KUKA KRL program: MyProgram_108().src

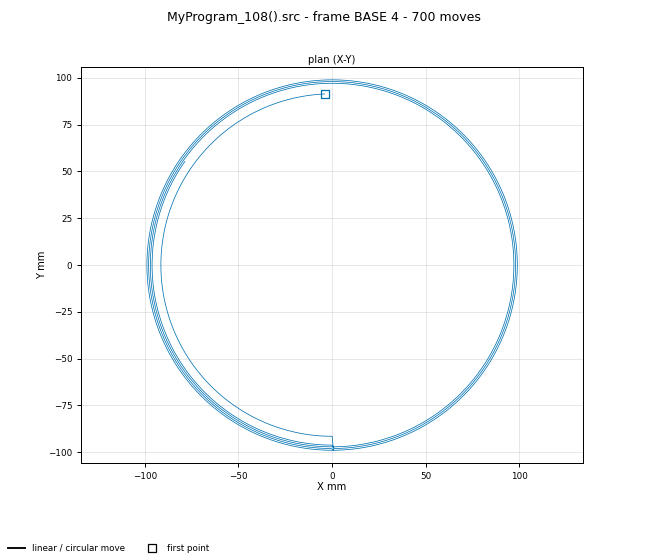
[picture p0: tool path of MyProgram_108().src in frame BASE 4, 700 of 700 moves have a stored position in this frame; points joined in program order, loops and branches not executed]
&ACCESS RVP
&REL 1
&PARAM TEMPLATE = C:\KRC\Roboter\Template\vorgabe
&PARAM EDITMASK = *
DEF MyProgram_108()
; ---- Setting reference (Base) ----
$BASE = BASE_DATA[4]

; --------------------------
; ---- Setting tool (TCP) ----
$TOOL = TOOL_DATA[3]
; --------------------------

$VEL.CP = VEL_APROX_PRINT
Startdeposition()
$VEL.CP = VEL_PRINT
LIN {X -4.0238,Y 91.3698,Z 95,A 87.6224,B 24.9054,C -2.2454,E1 24.992,E2 357.3815} C_DIS
LIN {X -6.9147,Y 91.1973,Z 95,A 89.45,B 24.9054,C -2.2451,E1 24.9869,E2 355.554} C_DIS
LIN {X -9.3244,Y 90.982,Z 95,A 91.0021,B 24.9054,C -2.2455,E1 24.9826,E2 354} C_DIS
LIN {X -12.2843,Y 90.6312,Z 95,A 92.9246,B 24.9054,C -2.2462,E1 24.9773,E2 352.0746} C_DIS
LIN {X -15.2613,Y 90.1762,Z 95,A 94.7056,B 24.9058,C -2.2414,E1 24.9724,E2 350.3032} C_DIS
LIN {X -18.2109,Y 89.6272,Z 95,A 96.5328,B 24.906,C -2.2382,E1 24.9674,E2 348.4816} C_DIS
LIN {X -20.6734,Y 89.0912,Z 95,A 98.1962,B 24.906,C -2.2396,E1 24.9628,E2 346.8129} C_DIS
LIN {X -23.8987,Y 88.2807,Z 95,A 100.2948,B 24.906,C -2.238,E1 24.9572,E2 344.715} C_DIS
LIN {X -26.5206,Y 87.5304,Z 95,A 102.081,B 24.906,C -2.2386,E1 24.9524,E2 342.9244} C_DIS
LIN {X -29.3987,Y 86.6047,Z 95,A 103.8698,B 24.9065,C -2.233,E1 24.9476,E2 341.1456} C_DIS
LIN {X -32.2068,Y 85.6002,Z 95,A 105.7005,B 24.9068,C -2.2294,E1 24.9429,E2 339.3198} C_DIS
LIN {X -34.3185,Y 84.7756,Z 95,A 107.1121,B 24.907,C -2.2272,E1 24.9392,E2 337.9104} C_DIS
LIN {X -36.7249,Y 83.7613,Z 95,A 108.969,B 24.9066,C -2.2318,E1 24.9344,E2 336.038} C_DIS
LIN {X -39.7684,Y 82.3598,Z 95,A 110.9169,B 24.9072,C -2.2238,E1 24.9295,E2 334.1043} C_DIS
LIN {X -42.0959,Y 81.1963,Z 95,A 112.6486,B 24.9072,C -2.2243,E1 24.9252,E2 332.3667} C_DIS
LIN {X -44.3837,Y 79.9673,Z 95,A 114.2579,B 24.9075,C -2.221,E1 24.9213,E2 330.7607} C_DIS
LIN {X -47.031,Y 78.4412,Z 95,A 116.0516,B 24.9081,C -2.2137,E1 24.917,E2 328.9788} C_DIS
LIN {X -48.938,Y 77.2658,Z 95,A 117.4609,B 24.9083,C -2.2113,E1 24.9136,E2 327.5709} C_DIS
LIN {X -50.8158,Y 76.044,Z 95,A 118.8703,B 24.9085,C -2.2088,E1 24.9104,E2 326.1629} C_DIS
LIN {X -52.965,Y 74.5612,Z 95,A 120.6248,B 24.9085,C -2.2093,E1 24.9063,E2 324.4013} C_DIS
LIN {X -55.6722,Y 72.5622,Z 95,A 122.7413,B 24.9088,C -2.2051,E1 24.9016,E2 322.287} C_DIS
LIN {X -58.1699,Y 70.5764,Z 95,A 124.7763,B 24.9091,C -2.2019,E1 24.8972,E2 320.2521} C_DIS
LIN {X -60.5846,Y 68.516,Z 95,A 126.8574,B 24.9091,C -2.2003,E1 24.8928,E2 318.1667} C_DIS
LIN {X -63.0597,Y 66.2451,Z 95,A 128.9712,B 24.9096,C -2.1956,E1 24.8885,E2 316.0552} C_DIS
LIN {X -65.4493,Y 63.8852,Z 95,A 131.0907,B 24.91,C -2.191,E1 24.8843,E2 313.9377} C_DIS
LIN {X -67.7678,Y 61.4204,Z 95,A 133.2194,B 24.9104,C -2.186,E1 24.8803,E2 311.8115} C_DIS
LIN {X -69.9777,Y 58.8902,Z 95,A 135.335,B 24.9108,C -2.181,E1 24.8765,E2 309.6983} C_DIS
LIN {X -72.0929,Y 56.2809,Z 95,A 137.4,B 24.9113,C -2.1742,E1 24.8729,E2 307.6397} C_DIS
LIN {X -73.682,Y 54.1815,Z 95,A 139.0043,B 24.9118,C -2.1684,E1 24.8702,E2 306.0416} C_DIS
LIN {X -75.623,Y 51.4376,Z 95,A 141.012,B 24.9125,C -2.1597,E1 24.8671,E2 304.0448} C_DIS
LIN {X -76.8604,Y 49.5696,Z 95,A 142.4242,B 24.9128,C -2.156,E1 24.8649,E2 302.6342} C_DIS
LIN {X -78.3252,Y 47.2218,Z 95,A 144.3699,B 24.9127,C -2.1575,E1 24.862,E2 300.6749} C_DIS
LIN {X -79.9567,Y 44.4027,Z 95,A 146.4407,B 24.9131,C -2.1526,E1 24.8592,E2 298.6051} C_DIS
LIN {X -81.3588,Y 41.778,Z 95,A 148.0983,B 24.914,C -2.1408,E1 24.8571,E2 296.9667} C_DIS
LIN {X -82.3563,Y 39.7757,Z 95,A 149.6193,B 24.914,C -2.1403,E1 24.8552,E2 295.4387} C_DIS
LIN {X -83.7601,Y 36.7275,Z 95,A 151.7374,B 24.9146,C -2.1345,E1 24.8528,E2 293.323} C_DIS
LIN {X -84.9155,Y 33.9747,Z 95,A 153.5097,B 24.9152,C -2.1258,E1 24.8509,E2 291.5616} C_DIS
LIN {X -85.8476,Y 31.5416,Z 95,A 155.2735,B 24.9153,C -2.1248,E1 24.8492,E2 289.7902} C_DIS
LIN {X -86.8443,Y 28.6883,Z 95,A 157.2742,B 24.9155,C -2.1221,E1 24.8474,E2 287.7845} C_DIS
LIN {X -87.8446,Y 25.4609,Z 95,A 159.1895,B 24.9165,C -2.1094,E1 24.8459,E2 285.8885} C_DIS
LIN {X -88.5337,Y 22.9445,Z 95,A 160.8359,B 24.9169,C -2.1047,E1 24.8447,E2 284.2438} C_DIS
LIN {X -89.154,Y 20.4015,Z 95,A 162.5816,B 24.9171,C -2.1027,E1 24.8435,E2 282.4927} C_DIS
LIN {X -89.7713,Y 17.4864,Z 95,A 164.4831,B 24.9175,C -2.0978,E1 24.8425,E2 280.5916} C_DIS
LIN {X -90.2986,Y 14.5298,Z 95,A 166.4559,B 24.9177,C -2.0945,E1 24.8416,E2 278.6149} C_DIS
LIN {X -90.677,Y 11.931,Z 95,A 167.9188,B 24.9186,C -2.0838,E1 24.841,E2 277.1689} C_DIS
LIN {X -90.9812,Y 9.3323,Z 95,A 169.7863,B 24.9184,C -2.0854,E1 24.8405,E2 275.2863} C_DIS
LIN {X -91.2368,Y 6.3646,Z 95,A 171.5613,B 24.9191,C -2.0766,E1 24.8401,E2 273.5216} C_DIS
LIN {X -91.3974,Y 3.3826,Z 95,A 173.3436,B 24.9198,C -2.068,E1 24.8399,E2 271.7493} C_DIS
LIN {X -91.4559,Y 0.6849,Z 95,A 175.1899,B 24.9198,C -2.0673,E1 24.8398,E2 269.8934} C_DIS
LIN {X -91.4213,Y -2.6095,Z 95,A 177.226,B 24.9204,C -2.0598,E1 24.8398,E2 267.8629} C_DIS
LIN {X -91.2891,Y -5.5881,Z 95,A 178.9966,B 24.9211,C -2.0509,E1 24.8402,E2 266.1029} C_DIS
LIN {X -91.092,Y -8.1813,Z 95,A -179.2539,B 24.9212,C -2.0494,E1 24.8406,E2 264.3466} C_DIS
LIN {X -90.7722,Y -11.1963,Z 95,A -177.45,B 24.9219,C -2.0405,E1 24.8411,E2 262.5531} C_DIS
LIN {X -90.4152,Y -13.7756,Z 95,A -175.6959,B 24.922,C -2.0391,E1 24.8418,E2 260.7919} C_DIS
LIN {X -89.8677,Y -16.9857,Z 95,A -173.7041,B 24.9226,C -2.0313,E1 24.8428,E2 258.8069} C_DIS
LIN {X -89.3965,Y -19.3113,Z 95,A -172.2569,B 24.9231,C -2.0255,E1 24.8436,E2 257.365} C_DIS
LIN {X -88.8068,Y -21.8634,Z 95,A -170.388,B 24.9229,C -2.0274,E1 24.8449,E2 255.4806} C_DIS
LIN {X -87.9436,Y -25.1114,Z 95,A -168.2536,B 24.9233,C -2.0219,E1 24.8465,E2 253.3469} C_DIS
LIN {X -86.9741,Y -28.287,Z 95,A -166.3203,B 24.9242,C -2.0112,E1 24.8481,E2 251.428} C_DIS
LIN {X -85.9537,Y -31.2506,Z 95,A -164.3287,B 24.9245,C -2.0062,E1 24.8499,E2 249.4369} C_DIS
LIN {X -84.7924,Y -34.2772,Z 95,A -162.3782,B 24.9252,C -1.9979,E1 24.8519,E2 247.4954} C_DIS
LIN {X -83.7612,Y -36.725,Z 95,A -160.48,B 24.925,C -2.0003,E1 24.854,E2 245.581} C_DIS
LIN {X -82.3569,Y -39.7745,Z 95,A -158.5243,B 24.9258,C -1.9899,E1 24.8563,E2 243.6396} C_DIS
LIN {X -81.1905,Y -42.1074,Z 95,A -156.7702,B 24.9258,C -1.989,E1 24.8586,E2 241.8781} C_DIS
LIN {X -79.9424,Y -44.4283,Z 95,A -155.1647,B 24.9263,C -1.9832,E1 24.8607,E2 240.278} C_DIS
LIN {X -78.4484,Y -47.019,Z 95,A -153.3895,B 24.9269,C -1.9752,E1 24.8632,E2 238.5128} C_DIS
LIN {X -77.2616,Y -48.9446,Z 95,A -151.9685,B 24.9271,C -1.9716,E1 24.8653,E2 237.093} C_DIS
LIN {X -76.0454,Y -50.8137,Z 95,A -150.5605,B 24.9274,C -1.9684,E1 24.8675,E2 235.6856} C_DIS
LIN {X -74.5698,Y -52.9529,Z 95,A -148.8116,B 24.9274,C -1.9681,E1 24.8703,E2 233.9288} C_DIS
LIN {X -72.467,Y -55.7958,Z 95,A -146.5187,B 24.9276,C -1.9651,E1 24.8742,E2 231.6319} C_DIS
LIN {X -70.3336,Y -58.4621,Z 95,A -144.434,B 24.9281,C -1.9584,E1 24.8778,E2 229.5536} C_DIS
LIN {X -68.1382,Y -61.0067,Z 95,A -142.3198,B 24.9284,C -1.9539,E1 24.8817,E2 227.4405} C_DIS
LIN {X -65.8506,Y -63.4691,Z 95,A -140.204,B 24.9287,C -1.9496,E1 24.8858,E2 225.3258} C_DIS
LIN {X -63.474,Y -65.8459,Z 95,A -138.0877,B 24.929,C -1.9456,E1 24.89,E2 223.2102} C_DIS
LIN {X -60.9908,Y -68.1525,Z 95,A -135.9582,B 24.9293,C -1.9415,E1 24.8944,E2 221.0817} C_DIS
LIN {X -58.4524,Y -70.3416,Z 95,A -133.8322,B 24.9296,C -1.9384,E1 24.8989,E2 218.9551} C_DIS
LIN {X -55.8153,Y -72.4519,Z 95,A -131.7259,B 24.9299,C -1.9342,E1 24.9035,E2 216.8509} C_DIS
LIN {X -53.5848,Y -74.1188,Z 95,A -129.9248,B 24.9299,C -1.933,E1 24.9076,E2 215.0463} C_DIS
LIN {X -51.4624,Y -75.6062,Z 95,A -128.4555,B 24.9305,C -1.9255,E1 24.9109,E2 213.59} C_DIS
LIN {X -49.6142,Y -76.8318,Z 95,A -127.0642,B 24.9306,C -1.9234,E1 24.9142,E2 212.1992} C_DIS
LIN {X -47.6627,Y -78.0572,Z 95,A -125.4981,B 24.9306,C -1.9252,E1 24.9179,E2 210.624} C_DIS
LIN {X -45.086,Y -79.5751,Z 95,A -123.5397,B 24.9306,C -1.9252,E1 24.9227,E2 208.6596} C_DIS
LIN {X -42.7806,Y -80.8361,Z 95,A -122.0791,B 24.9311,C -1.9171,E1 24.9262,E2 207.2143} C_DIS
LIN {X -40.6274,Y -81.9393,Z 95,A -120.4471,B 24.931,C -1.919,E1 24.9303,E2 205.5733} C_DIS
LIN {X -38.0993,Y -83.1467,Z 95,A -118.6241,B 24.931,C -1.9192,E1 24.935,E2 203.7454} C_DIS
LIN {X -35.3431,Y -84.3536,Z 95,A -116.8551,B 24.9314,C -1.9134,E1 24.9395,E2 201.9859} C_DIS
LIN {X -32.8352,Y -85.3622,Z 95,A -115.0915,B 24.9314,C -1.9141,E1 24.9441,E2 200.2169} C_DIS
LIN {X -30.4684,Y -86.2342,Z 95,A -113.6232,B 24.9317,C -1.909,E1 24.9479,E2 198.7577} C_DIS
LIN {X -27.9724,Y -87.0759,Z 95,A -111.9226,B 24.9317,C -1.9094,E1 24.9524,E2 197.0531} C_DIS
LIN {X -25.1205,Y -87.9411,Z 95,A -109.9953,B 24.9317,C -1.9101,E1 24.9576,E2 195.1209} C_DIS
LIN {X -21.8609,Y -88.8075,Z 95,A -107.8812,B 24.9317,C -1.9089,E1 24.9633,E2 193.0065} C_DIS
LIN {X -18.9546,Y -89.4743,Z 95,A -105.9637,B 24.9317,C -1.9097,E1 24.9686,E2 191.0848} C_DIS
LIN {X -15.8541,Y -90.0744,Z 95,A -104.121,B 24.932,C -1.9045,E1 24.9736,E2 189.2526} C_DIS
LIN {X -13.1259,Y -90.5119,Z 95,A -102.2258,B 24.9316,C -1.9095,E1 24.9789,E2 187.3437} C_DIS
LIN {X -9.6461,Y -90.9483,Z 95,A -100.1452,B 24.9319,C -1.9053,E1 24.9846,E2 185.2718} C_DIS
LIN {X -6.6432,Y -91.218,Z 95,A -98.113,B 24.9316,C -1.9101,E1 24.9903,E2 183.2274} C_DIS
LIN {X -3.0457,Y -91.4079,Z 95,A -95.8652,B 24.9316,C -1.9101,E1 24.9966,E2 180.9792} C_DIS
LIN {X 0.0472,Y -91.4598,Z 95,A -93.9773,B 24.9317,C -1.9087,E1 25.0018,E2 179.0946} C_DIS
LIN {X 0.0472,Y -91.4598,Z 95,A -93.9773,B 24.9317,C -1.9087,E1 25.0018,E2 179.0946} C_DIS
Enddeposition()
LIN {X 0.6782,Y -98.9101,Z 96,A -93.6566,B 24.9403,C -1.7848,E1 25.0019,E2 179.0676} C_DIS
Startdeposition()
$VEL.CP = VEL_PRINT
LIN {X 3.095,Y -98.8665,Z 96,A -92.0066,B 24.9396,C -1.7945,E1 25.0066,E2 177.3949} C_DIS
LIN {X 6.0657,Y -98.7307,Z 96,A -90.1754,B 24.9393,C -1.7993,E1 25.0117,E2 175.5531} C_DIS
LIN {X 9.2855,Y -98.4783,Z 96,A -88.4513,B 24.9396,C -1.7947,E1 25.0165,E2 173.8407} C_DIS
LIN {X 12.1085,Y -98.1729,Z 96,A -86.8644,B 24.9397,C -1.7935,E1 25.0209,E2 172.2578} C_DIS
LIN {X 15.0538,Y -97.7627,Z 96,A -85.1441,B 24.9397,C -1.7947,E1 25.0256,E2 170.5364} C_DIS
LIN {X 17.5683,Y -97.3423,Z 96,A -83.58,B 24.9393,C -1.7991,E1 25.03,E2 168.9634} C_DIS
LIN {X 21.0203,Y -96.6557,Z 96,A -81.6027,B 24.9393,C -1.7986,E1 25.0353,E2 166.9899} C_DIS
LIN {X 24.0348,Y -95.9524,Z 96,A -79.6458,B 24.9388,C -1.8066,E1 25.0407,E2 165.0169} C_DIS
LIN {X 26.9078,Y -95.1848,Z 96,A -78.0952,B 24.9391,C -1.8019,E1 25.0448,E2 163.4799} C_DIS
LIN {X 29.8735,Y -94.298,Z 96,A -76.1387,B 24.9386,C -1.8102,E1 25.0501,E2 161.5073} C_DIS
LIN {X 32.909,Y -93.2802,Z 96,A -74.3585,B 24.9386,C -1.8097,E1 25.0548,E2 159.7317} C_DIS
LIN {X 36.1079,Y -92.089,Z 96,A -72.5177,B 24.9388,C -1.8072,E1 25.0596,E2 157.9009} C_DIS
LIN {X 38.357,Y -91.1751,Z 96,A -71.0343,B 24.9384,C -1.8122,E1 25.0634,E2 156.4091} C_DIS
LIN {X 41.1919,Y -89.932,Z 96,A -69.129,B 24.938,C -1.8193,E1 25.0683,E2 154.4918} C_DIS
LIN {X 43.8758,Y -88.6515,Z 96,A -67.6123,B 24.9383,C -1.8141,E1 25.0721,E2 152.9914} C_DIS
LIN {X 46.0382,Y -87.548,Z 96,A -66.1791,B 24.9381,C -1.8175,E1 25.0756,E2 151.554} C_DIS
LIN {X 48.7559,Y -86.0662,Z 96,A -64.4251,B 24.938,C -1.8191,E1 25.0799,E2 149.8014} C_DIS
LIN {X 51.32,Y -84.5602,Z 96,A -62.677,B 24.9377,C -1.8233,E1 25.0841,E2 148.0487} C_DIS
LIN {X 53.9418,Y -82.9145,Z 96,A -60.9235,B 24.9376,C -1.8252,E1 25.0882,E2 146.2965} C_DIS
LIN {X 56.4088,Y -81.2541,Z 96,A -59.1765,B 24.9373,C -1.8296,E1 25.0923,E2 144.5449} C_DIS
LIN {X 58.9247,Y -79.4507,Z 96,A -57.4236,B 24.9371,C -1.8318,E1 25.0962,E2 142.7932} C_DIS
LIN {X 61.2852,Y -77.6421,Z 96,A -55.7092,B 24.9369,C -1.8352,E1 25.1,E2 141.077} C_DIS
LIN {X 63.2658,Y -76.0369,Z 96,A -54.1499,B 24.9364,C -1.8417,E1 25.1034,E2 139.5082} C_DIS
LIN {X 65.5606,Y -74.0694,Z 96,A -52.5233,B 24.9364,C -1.8408,E1 25.1068,E2 137.8902} C_DIS
LIN {X 67.7207,Y -72.0977,Z 96,A -50.812,B 24.9362,C -1.8455,E1 25.1103,E2 136.1747} C_DIS
LIN {X 69.4696,Y -70.414,Z 96,A -49.3807,B 24.9359,C -1.8499,E1 25.1132,E2 134.7391} C_DIS
LIN {X 71.6402,Y -68.2071,Z 96,A -47.4301,B 24.9351,C -1.8605,E1 25.117,E2 132.7717} C_DIS
LIN {X 73.6644,Y -66.0131,Z 96,A -45.9132,B 24.9354,C -1.8565,E1 25.1198,E2 131.271} C_DIS
LIN {X 75.2548,Y -64.1941,Z 96,A -44.5178,B 24.9352,C -1.86,E1 25.1224,E2 129.8737} C_DIS
LIN {X 76.8842,Y -62.2333,Z 96,A -42.96,B 24.9347,C -1.8671,E1 25.1252,E2 128.3064} C_DIS
LIN {X 78.7216,Y -59.8952,Z 96,A -41.1378,B 24.934,C -1.8757,E1 25.1283,E2 126.4725} C_DIS
LIN {X 80.485,Y -57.5007,Z 96,A -39.5926,B 24.9342,C -1.8733,E1 25.1308,E2 124.9403} C_DIS
LIN {X 82.2463,Y -54.9552,Z 96,A -37.6432,B 24.9334,C -1.8846,E1 25.1339,E2 122.9741} C_DIS
LIN {X 84.1104,Y -52.0554,Z 96,A -35.8438,B 24.9336,C -1.8824,E1 25.1365,E2 121.189} C_DIS
LIN {X 85.7335,Y -49.3349,Z 96,A -34.0023,B 24.9332,C -1.8879,E1 25.1391,E2 119.3437} C_DIS
LIN {X 87.2368,Y -46.6291,Z 96,A -32.2525,B 24.9329,C -1.8914,E1 25.1415,E2 117.5948} C_DIS
LIN {X 88.5134,Y -44.1543,Z 96,A -30.5576,B 24.9324,C -1.8995,E1 25.1436,E2 115.8899} C_DIS
LIN {X 89.932,Y -41.1919,Z 96,A -28.5607,B 24.9317,C -1.909,E1 25.146,E2 113.8814} C_DIS
LIN {X 91.1751,Y -38.357,Z 96,A -26.8891,B 24.9317,C -1.9096,E1 25.1478,E2 112.2174} C_DIS
LIN {X 92.4821,Y -35.089,Z 96,A -24.9212,B 24.9314,C -1.9131,E1 25.1498,E2 110.2523} C_DIS
LIN {X 93.5365,Y -32.1787,Z 96,A -22.9733,B 24.9305,C -1.9249,E1 25.1517,E2 108.2876} C_DIS
LIN {X 94.4597,Y -29.3519,Z 96,A -21.4616,B 24.9308,C -1.9218,E1 25.1529,E2 106.7917} C_DIS
LIN {X 95.255,Y -26.6598,Z 96,A -19.8173,B 24.9303,C -1.9277,E1 25.1542,E2 105.143} C_DIS
LIN {X 95.9524,Y -24.0348,Z 96,A -18.0851,B 24.9295,C -1.939,E1 25.1554,E2 103.3939} C_DIS
LIN {X 96.6557,Y -21.0203,Z 96,A -16.4138,B 24.9295,C -1.9399,E1 25.1564,E2 101.7304} C_DIS
LIN {X 97.3423,Y -17.5683,Z 96,A -14.3925,B 24.929,C -1.9457,E1 25.1575,E2 99.7071} C_DIS
LIN {X 97.8462,Y -14.5141,Z 96,A -12.4852,B 24.9283,C -1.956,E1 25.1583,E2 97.7867} C_DIS
LIN {X 98.3141,Y -10.9028,Z 96,A -10.4044,B 24.9279,C -1.9617,E1 25.159,E2 95.7048} C_DIS
LIN {X 98.6053,Y -7.8211,Z 96,A -8.7334,B 24.9278,C -1.9626,E1 25.1594,E2 94.0416} C_DIS
LIN {X 98.8211,Y -4.3081,Z 96,A -6.7984,B 24.9276,C -1.965,E1 25.1597,E2 92.1125} C_DIS
LIN {X 98.8993,Y -1.7598,Z 96,A -5.2454,B 24.927,C -1.9728,E1 25.1597,E2 90.5502} C_DIS
LIN {X 98.8993,Y 1.7598,Z 96,A -3.2752,B 24.9267,C -1.9766,E1 25.1597,E2 88.5828} C_DIS
LIN {X 98.7977,Y 4.8536,Z 96,A -1.3274,B 24.9259,C -1.9886,E1 25.1595,E2 86.6183} C_DIS
LIN {X 98.5956,Y 7.9425,Z 96,A 0.3785,B 24.9257,C -1.9908,E1 25.1592,E2 84.9173} C_DIS
LIN {X 98.2506,Y 11.4452,Z 96,A 2.3109,B 24.9255,C -1.993,E1 25.1586,E2 82.9911} C_DIS
LIN {X 97.8462,Y 14.5141,Z 96,A 4.2589,B 24.9246,C -2.0049,E1 25.1578,E2 81.0266} C_DIS
LIN {X 97.3423,Y 17.5683,Z 96,A 5.9301,B 24.9246,C -2.0056,E1 25.157,E2 79.3634} C_DIS
LIN {X 96.6557,Y 21.0203,Z 96,A 7.8978,B 24.9243,C -2.0091,E1 25.1559,E2 77.399} C_DIS
LIN {X 95.9524,Y 24.0348,Z 96,A 9.8459,B 24.9234,C -2.0208,E1 25.1546,E2 75.4345} C_DIS
LIN {X 95.1516,Y 27.0249,Z 96,A 11.5174,B 24.9234,C -2.0215,E1 25.1534,E2 73.7712} C_DIS
LIN {X 94.298,Y 29.8735,Z 96,A 13.1393,B 24.9233,C -2.0226,E1 25.152,E2 72.1558} C_DIS
LIN {X 93.3556,Y 32.6939,Z 96,A 14.8826,B 24.9228,C -2.0286,E1 25.1505,E2 70.4081} C_DIS
LIN {X 92.2887,Y 35.5997,Z 96,A 16.6325,B 24.9226,C -2.0321,E1 25.1487,E2 68.6598} C_DIS
LIN {X 91.1751,Y 38.357,Z 96,A 18.3438,B 24.9222,C -2.0367,E1 25.1469,E2 66.9471} C_DIS
LIN {X 90.2064,Y 40.583,Z 96,A 19.7417,B 24.9219,C -2.0404,E1 25.1453,E2 65.5481} C_DIS
LIN {X 89.1832,Y 42.7846,Z 96,A 21.1714,B 24.9216,C -2.0453,E1 25.1436,E2 64.1145} C_DIS
LIN {X 87.8025,Y 45.555,Z 96,A 23.121,B 24.9207,C -2.0564,E1 25.1411,E2 62.149} C_DIS
LIN {X 86.3918,Y 48.1728,Z 96,A 24.7172,B 24.9207,C -2.0561,E1 25.139,E2 60.5618} C_DIS
LIN {X 84.8438,Y 50.8534,Z 96,A 26.616,B 24.92,C -2.0651,E1 25.1363,E2 58.6517} C_DIS
LIN {X 83.2095,Y 53.4823,Z 96,A 28.2889,B 24.92,C -2.0651,E1 25.1338,E2 56.9873} C_DIS
LIN {X 81.2541,Y 56.4088,Z 96,A 30.2269,B 24.92,C -2.0663,E1 25.1308,E2 55.0559} C_DIS
LIN {X 79.8328,Y 58.4028,Z 96,A 31.664,B 24.9196,C -2.0705,E1 25.1284,E2 53.6157} C_DIS
LIN {X 77.9807,Y 60.8567,Z 96,A 33.4093,B 24.9194,C -2.0734,E1 25.1255,E2 51.8718} C_DIS
LIN {X 76.4637,Y 62.7522,Z 96,A 35.0079,B 24.9185,C -2.0843,E1 25.1226,E2 50.255} C_DIS
LIN {X 74.5415,Y 65.0211,Z 96,A 36.5222,B 24.9189,C -2.0801,E1 25.1199,E2 48.7574} C_DIS
LIN {X 72.9233,Y 66.8308,Z 96,A 37.9536,B 24.9185,C -2.0843,E1 25.1172,E2 47.3224} C_DIS
LIN {X 70.7978,Y 69.0811,Z 96,A 39.7062,B 24.9184,C -2.0866,E1 25.1138,E2 45.5721} C_DIS
LIN {X 69.0811,Y 70.7978,Z 96,A 41.1059,B 24.9181,C -2.0893,E1 25.111,E2 44.1717} C_DIS
LIN {X 66.9205,Y 72.841,Z 96,A 42.853,B 24.9178,C -2.0938,E1 25.1075,E2 42.4212} C_DIS
LIN {X 64.6098,Y 74.9007,Z 96,A 44.6459,B 24.9175,C -2.0973,E1 25.1037,E2 40.6271} C_DIS
LIN {X 62.7522,Y 76.4637,Z 96,A 46.2064,B 24.9168,C -2.1059,E1 25.1003,E2 39.0522} C_DIS
LIN {X 60.4242,Y 78.314,Z 96,A 47.7948,B 24.917,C -2.1039,E1 25.0968,E2 37.4743} C_DIS
LIN {X 57.9453,Y 80.1678,Z 96,A 49.5086,B 24.917,C -2.1039,E1 25.093,E2 35.7665} C_DIS
LIN {X 55.9604,Y 81.5657,Z 96,A 50.9099,B 24.9168,C -2.1062,E1 25.0898,E2 34.365} C_DIS
LIN {X 53.4823,Y 83.2095,Z 96,A 52.686,B 24.9164,C -2.111,E1 25.0856,E2 32.5833} C_DIS
LIN {X 50.7519,Y 84.9037,Z 96,A 54.527,B 24.9163,C -2.113,E1 25.0812,E2 30.7433} C_DIS
LIN {X 48.1728,Y 86.3918,Z 96,A 56.2909,B 24.916,C -2.1169,E1 25.0769,E2 28.9753} C_DIS
LIN {X 45.555,Y 87.8025,Z 96,A 58.1186,B 24.9155,C -2.1232,E1 25.0724,E2 27.1379} C_DIS
LIN {X 42.7846,Y 89.1832,Z 96,A 59.7968,B 24.9156,C -2.1211,E1 25.0682,E2 25.4692} C_DIS
LIN {X 40.0852,Y 90.4307,Z 96,A 61.425,B 24.9158,C -2.1194,E1 25.0641,E2 23.8489} C_DIS
LIN {X 37.348,Y 91.5931,Z 96,A 63.2176,B 24.9154,C -2.1239,E1 25.0594,E2 22.0498} C_DIS
LIN {X 34.4645,Y 92.7186,Z 96,A 65.1333,B 24.9149,C -2.1302,E1 25.0544,E2 20.1234} C_DIS
LIN {X 31.5458,Y 93.7498,Z 96,A 66.8126,B 24.9151,C -2.1275,E1 25.05,E2 18.4537} C_DIS
LIN {X 28.1905,Y 94.8128,Z 96,A 68.7905,B 24.9151,C -2.1268,E1 25.0447,E2 16.4811} C_DIS
LIN {X 25.2105,Y 95.6502,Z 96,A 70.749,B 24.9146,C -2.1341,E1 25.0394,E2 14.5085} C_DIS
LIN {X 22.3235,Y 96.363,Z 96,A 72.3014,B 24.915,C -2.1288,E1 25.0352,E2 12.9709} C_DIS
LIN {X 19.2977,Y 97.0161,Z 96,A 74.2607,B 24.9145,C -2.1357,E1 25.0298,E2 10.9976} C_DIS
LIN {X 16.2523,Y 97.5706,Z 96,A 75.9419,B 24.9147,C -2.1323,E1 25.0252,E2 9.3264} C_DIS
LIN {X 12.7708,Y 98.0871,Z 96,A 77.9631,B 24.9147,C -2.1321,E1 25.0197,E2 7.3073} C_DIS
LIN {X 9.6955,Y 98.4405,Z 96,A 79.8829,B 24.9143,C -2.137,E1 25.0143,E2 5.3772} C_DIS
LIN {X 6.7319,Y 98.6856,Z 96,A 81.4367,B 24.9148,C -2.1309,E1 25.01,E2 3.8385} C_DIS
LIN {X 3.6409,Y 98.8498,Z 96,A 83.1975,B 24.9149,C -2.1296,E1 25.0051,E2 2.0813} C_DIS
LIN {X 0.6678,Y 98.9127,Z 96,A 84.9532,B 24.9149,C -2.1306,E1 25.0002,E2 0.3236} C_DIS
LIN {X -2.4275,Y 98.887,Z 96,A 86.7149,B 24.9149,C -2.129,E1 24.9953,E2 -1.4344} C_DIS
LIN {X -5.3989,Y 98.7675,Z 96,A 88.4711,B 24.9149,C -2.1297,E1 24.9904,E2 -3.1926} C_DIS
LIN {X -8.4868,Y 98.5521,Z 96,A 90.4345,B 24.9145,C -2.135,E1 24.9849,E2 -5.1695} C_DIS
LIN {X -11.5661,Y 98.2364,Z 96,A 92.1189,B 24.9149,C -2.1301,E1 24.9802,E2 -6.8434} C_DIS
LIN {X -15.0538,Y 97.7627,Z 96,A 94.0705,B 24.9153,C -2.1257,E1 24.9749,E2 -8.786} C_DIS
LIN {X -17.5683,Y 97.3423,Z 96,A 95.64,B 24.9151,C -2.1279,E1 24.9705,E2 -10.3623} C_DIS
LIN {X -21.0203,Y 96.6557,Z 96,A 97.6246,B 24.9154,C -2.1242,E1 24.9651,E2 -12.3406} C_DIS
LIN {X -24.0348,Y 95.9524,Z 96,A 99.5901,B 24.915,C -2.1286,E1 24.9598,E2 -14.3192} C_DIS
LIN {X -26.9078,Y 95.1848,Z 96,A 101.1936,B 24.9155,C -2.1227,E1 24.9555,E2 -15.911} C_DIS
LIN {X -29.8735,Y 94.298,Z 96,A 102.9129,B 24.9159,C -2.118,E1 24.9509,E2 -17.6222} C_DIS
LIN {X -32.1787,Y 93.5365,Z 96,A 104.5242,B 24.9154,C -2.1235,E1 24.9466,E2 -19.2496} C_DIS
LIN {X -35.089,Y 92.4821,Z 96,A 106.2116,B 24.9159,C -2.1175,E1 24.9422,E2 -20.9262} C_DIS
LIN {X -37.8538,Y 91.3872,Z 96,A 107.8487,B 24.9163,C -2.1121,E1 24.938,E2 -22.5541} C_DIS
LIN {X -40.0852,Y 90.4307,Z 96,A 109.32,B 24.9163,C -2.1123,E1 24.9342,E2 -24.0294} C_DIS
LIN {X -42.7846,Y 89.1832,Z 96,A 110.9877,B 24.9167,C -2.1078,E1 24.93,E2 -25.6905} C_DIS
LIN {X -44.9604,Y 88.1064,Z 96,A 112.3992,B 24.9168,C -2.1057,E1 24.9265,E2 -27.1008} C_DIS
LIN {X -47.2161,Y 86.9184,Z 96,A 113.9721,B 24.9168,C -2.1065,E1 24.9226,E2 -28.6801} C_DIS
LIN {X -49.8084,Y 85.4614,Z 96,A 115.8121,B 24.9168,C -2.1075,E1 24.9182,E2 -30.5279} C_DIS
LIN {X -52.4571,Y 83.8595,Z 96,A 117.5015,B 24.9172,C -2.1006,E1 24.9142,E2 -32.2062} C_DIS
LIN {X -54.9552,Y 82.2463,Z 96,A 119.3422,B 24.9172,C -2.1013,E1 24.9099,E2 -34.0547} C_DIS
LIN {X -57.5007,Y 80.485,Z 96,A 121.0324,B 24.9178,C -2.0942,E1 24.906,E2 -35.7337} C_DIS
LIN {X -59.8952,Y 78.7216,Z 96,A 122.8738,B 24.9178,C -2.0947,E1 24.9019,E2 -37.5828} C_DIS
LIN {X -62.2333,Y 76.8842,Z 96,A 124.4029,B 24.9185,C -2.0844,E1 24.8986,E2 -39.093} C_DIS
LIN {X -64.1941,Y 75.2548,Z 96,A 125.9775,B 24.9185,C -2.0844,E1 24.8952,E2 -40.6739} C_DIS
LIN {X -66.4285,Y 73.2925,Z 96,A 127.8198,B 24.9185,C -2.0845,E1 24.8914,E2 -42.5238} C_DIS
LIN {X -68.6003,Y 71.2612,Z 96,A 129.3494,B 24.9193,C -2.074,E1 24.8883,E2 -44.0345} C_DIS
LIN {X -70.4141,Y 69.4696,Z 96,A 130.9247,B 24.9193,C -2.0737,E1 24.8852,E2 -45.6159} C_DIS
LIN {X -72.841,Y 66.9205,Z 96,A 132.9165,B 24.9199,C -2.0671,E1 24.8814,E2 -47.6006} C_DIS
LIN {X -74.9007,Y 64.6098,Z 96,A 134.8891,B 24.9198,C -2.0686,E1 24.8778,E2 -49.5856} C_DIS
LIN {X -76.8075,Y 62.3279,Z 96,A 136.4194,B 24.9206,C -2.0576,E1 24.8751,E2 -51.097} C_DIS
LIN {X -78.314,Y 60.4242,Z 96,A 137.8337,B 24.9209,C -2.0542,E1 24.8727,E2 -52.5096} C_DIS
LIN {X -79.8452,Y 58.3858,Z 96,A 139.4103,B 24.9209,C -2.0535,E1 24.87,E2 -54.0924} C_DIS
LIN {X -81.8719,Y 55.5082,Z 96,A 141.4543,B 24.9213,C -2.0481,E1 24.8668,E2 -56.1335} C_DIS
LIN {X -83.5702,Y 52.9203,Z 96,A 143.3767,B 24.9213,C -2.0474,E1 24.8639,E2 -58.0638} C_DIS
LIN {X -85.1216,Y 50.3833,Z 96,A 144.9405,B 24.9222,C -2.0372,E1 24.8616,E2 -59.6114} C_DIS
LIN {X -86.6581,Y 47.6961,Z 96,A 146.9146,B 24.9222,C -2.038,E1 24.8589,E2 -61.5978} C_DIS
LIN {X -88.051,Y 45.0688,Z 96,A 148.4463,B 24.923,C -2.0266,E1 24.857,E2 -63.1104} C_DIS
LIN {X -89.1832,Y 42.7846,Z 96,A 150.0233,B 24.923,C -2.0255,E1 24.855,E2 -64.6935} C_DIS
LIN {X -90.6489,Y 39.5846,Z 96,A 152.0176,B 24.9236,C -2.0179,E1 24.8528,E2 -66.6806} C_DIS
LIN {X -91.8448,Y 36.7295,Z 96,A 153.9922,B 24.9236,C -2.0185,E1 24.8507,E2 -68.6674} C_DIS
LIN {X -92.9474,Y 33.8371,Z 96,A 155.6861,B 24.9243,C -2.0097,E1 24.849,E2 -70.35} C_DIS
LIN {X -94.0924,Y 30.5088,Z 96,A 157.6807,B 24.9249,C -2.0018,E1 24.8473,E2 -72.3372} C_DIS
LIN {X -95.0027,Y 27.5503,Z 96,A 159.4537,B 24.9253,C -1.9955,E1 24.8459,E2 -74.1054} C_DIS
LIN {X -95.7861,Y 24.6816,Z 96,A 161.2205,B 24.9256,C -1.9916,E1 24.8446,E2 -75.8731} C_DIS
LIN {X -96.5133,Y 21.6728,Z 96,A 163.1956,B 24.9256,C -1.9919,E1 24.8433,E2 -77.8606} C_DIS
LIN {X -97.1424,Y 18.6419,Z 96,A 164.8901,B 24.9263,C -1.983,E1 24.8424,E2 -79.5438} C_DIS
LIN {X -97.6607,Y 15.7137,Z 96,A 166.7362,B 24.9263,C -1.9815,E1 24.8416,E2 -81.3974} C_DIS
LIN {X -98.0871,Y 12.7707,Z 96,A 168.3013,B 24.9272,C -1.9708,E1 24.841,E2 -82.9462} C_DIS
LIN {X -98.4405,Y 9.6955,Z 96,A 170.2767,B 24.9272,C -1.9711,E1 24.8404,E2 -84.9341} C_DIS
LIN {X -98.6938,Y 6.6105,Z 96,A 171.9709,B 24.9278,C -1.962,E1 24.8401,E2 -86.6169} C_DIS
LIN {X -98.8665,Y 3.095,Z 96,A 173.9661,B 24.9284,C -1.954,E1 24.8398,E2 -88.605} C_DIS
LIN {X -98.9169,Y 0,Z 96,A 175.9444,B 24.9284,C -1.9544,E1 24.8398,E2 -90.5961} C_DIS
LIN {X -98.8665,Y -3.095,Z 96,A 177.6358,B 24.9291,C -1.9453,E1 24.8399,E2 -92.276} C_DIS
LIN {X -98.7293,Y -6.0851,Z 96,A 179.4847,B 24.9291,C -1.9436,E1 24.8402,E2 -94.1319} C_DIS
LIN {X -98.4907,Y -9.1518,Z 96,A -178.8239,B 24.9298,C -1.9349,E1 24.8406,E2 -95.8128} C_DIS
LIN {X -98.1729,Y -12.1085,Z 96,A -177.1805,B 24.9304,C -1.9268,E1 24.8411,E2 -97.4467} C_DIS
LIN {X -97.7627,Y -15.0538,Z 96,A -175.4457,B 24.9308,C -1.9218,E1 24.8418,E2 -99.1799} C_DIS
LIN {X -97.3423,Y -17.5683,Z 96,A -173.868,B 24.9308,C -1.9206,E1 24.8426,E2 -100.764} C_DIS
LIN {X -96.6557,Y -21.0203,Z 96,A -171.8069,B 24.9313,C -1.915,E1 24.8438,E2 -102.8239} C_DIS
LIN {X -95.8722,Y -24.3469,Z 96,A -169.8386,B 24.9317,C -1.9085,E1 24.8451,E2 -104.7883} C_DIS
LIN {X -95.1848,Y -26.9078,Z 96,A -168.3345,B 24.9321,C -1.9028,E1 24.8462,E2 -106.2875} C_DIS
LIN {X -94.298,Y -29.8735,Z 96,A -166.36,B 24.9321,C -1.9035,E1 24.8478,E2 -108.2751} C_DIS
LIN {X -93.3153,Y -32.8088,Z 96,A -164.6664,B 24.9327,C -1.8948,E1 24.8493,E2 -109.9576} C_DIS
LIN {X -92.089,Y -36.1079,Z 96,A -162.7053,B 24.9333,C -1.8863,E1 24.8513,E2 -111.9093} C_DIS
LIN {X -91.1751,Y -38.357,Z 96,A -161.2122,B 24.9333,C -1.8851,E1 24.8529,E2 -113.408} C_DIS
LIN {X -89.932,Y -41.1919,Z 96,A -159.284,B 24.9334,C -1.8846,E1 24.8551,E2 -115.3455} C_DIS
LIN {X -88.4676,Y -44.2467,Z 96,A -157.4879,B 24.9342,C -1.8735,E1 24.8573,E2 -117.1249} C_DIS
LIN {X -87.2368,Y -46.6291,Z 96,A -155.7469,B 24.9341,C -1.8756,E1 24.8596,E2 -118.8801} C_DIS
LIN {X -85.6655,Y -49.4533,Z 96,A -154.0104,B 24.9347,C -1.866,E1 24.8619,E2 -120.6028} C_DIS
LIN {X -84.2133,Y -51.8907,Z 96,A -152.4127,B 24.9351,C -1.8601,E1 24.8642,E2 -122.1946} C_DIS
LIN {X -82.6139,Y -54.3977,Z 96,A -150.6478,B 24.9354,C -1.8571,E1 24.8669,E2 -123.9613} C_DIS
LIN {X -80.8729,Y -56.9571,Z 96,A -148.8775,B 24.9357,C -1.8518,E1 24.8697,E2 -125.7277} C_DIS
LIN {X -79.1227,Y -59.3613,Z 96,A -147.0511,B 24.9357,C -1.8511,E1 24.8728,E2 -127.5614} C_DIS
LIN {X -77.228,Y -61.8091,Z 96,A -145.343,B 24.9363,C -1.8439,E1 24.8757,E2 -129.2604} C_DIS
LIN {X -75.6879,Y -63.6858,Z 96,A -143.9295,B 24.9365,C -1.8409,E1 24.8782,E2 -130.6731} C_DIS
LIN {X -74.0612,Y -65.5698,Z 96,A -142.5138,B 24.9368,C -1.8367,E1 24.8808,E2 -132.0853} C_DIS
LIN {X -72.0977,Y -67.7207,Z 96,A -140.7857,B 24.9369,C -1.8344,E1 24.8841,E2 -133.8155} C_DIS
LIN {X -70.414,Y -69.4696,Z 96,A -139.3401,B 24.937,C -1.8328,E1 24.8869,E2 -135.2634} C_DIS
LIN {X -68.2071,Y -71.6402,Z 96,A -137.37,B 24.9369,C -1.8352,E1 24.8909,E2 -137.2475} C_DIS
LIN {X -65.78,Y -73.873,Z 96,A -135.6123,B 24.9375,C -1.8261,E1 24.8945,E2 -138.9905} C_DIS
LIN {X -63.2658,Y -76.0369,Z 96,A -133.6907,B 24.9377,C -1.8224,E1 24.8986,E2 -140.9109} C_DIS
LIN {X -60.8567,Y -77.9807,Z 96,A -131.8253,B 24.9377,C -1.8217,E1 24.9027,E2 -142.7814} C_DIS
LIN {X -58.4841,Y -79.7733,Z 96,A -130.194,B 24.9382,C -1.8155,E1 24.9063,E2 -144.4039} C_DIS
LIN {X -56.4088,Y -81.2541,Z 96,A -128.6209,B 24.9382,C -1.8164,E1 24.9099,E2 -145.9845} C_DIS
LIN {X -53.4823,Y -83.2095,Z 96,A -126.6659,B 24.9386,C -1.8103,E1 24.9145,E2 -147.9313} C_DIS
LIN {X -51.32,Y -84.5602,Z 96,A -125.0936,B 24.9385,C -1.8115,E1 24.9182,E2 -149.5113} C_DIS
LIN {X -48.7559,Y -86.0662,Z 96,A -123.2552,B 24.9384,C -1.8131,E1 24.9227,E2 -151.3591} C_DIS
LIN {X -46.0382,Y -87.548,Z 96,A -121.5676,B 24.9388,C -1.807,E1 24.9269,E2 -153.0369} C_DIS
LIN {X -43.3865,Y -88.894,Z 96,A -119.7297,B 24.9387,C -1.809,E1 24.9315,E2 -154.8844} C_DIS
LIN {X -40.694,Y -90.1563,Z 96,A -118.1064,B 24.939,C -1.8036,E1 24.9356,E2 -156.4987} C_DIS
LIN {X -37.8538,Y -91.3872,Z 96,A -116.4068,B 24.9394,C -1.7983,E1 24.9399,E2 -158.1898} C_DIS
LIN {X -35.089,Y -92.4821,Z 96,A -114.6482,B 24.9394,C -1.798,E1 24.9445,E2 -159.9514} C_DIS
LIN {X -32.1787,Y -93.5365,Z 96,A -112.6834,B 24.9391,C -1.8026,E1 24.9497,E2 -161.9311} C_DIS
LIN {X -29.0207,Y -94.5624,Z 96,A -110.9219,B 24.9396,C -1.7954,E1 24.9544,E2 -163.6784} C_DIS
LIN {X -25.9001,Y -95.4639,Z 96,A -109.0593,B 24.9397,C -1.7934,E1 24.9594,E2 -165.5394} C_DIS
LIN {X -23.386,Y -96.1107,Z 96,A -107.4774,B 24.9396,C -1.7955,E1 24.9637,E2 -167.1283} C_DIS
LIN {X -19.9519,Y -96.8818,Z 96,A -105.4945,B 24.9398,C -1.7925,E1 24.9691,E2 -169.1067} C_DIS
LIN {X -16.911,Y -97.4605,Z 96,A -103.7326,B 24.9398,C -1.7907,E1 24.9739,E2 -170.8661} C_DIS
LIN {X -13.9735,Y -97.923,Z 96,A -101.9768,B 24.9398,C -1.7915,E1 24.9788,E2 -172.6254} C_DIS
LIN {X -10.9028,Y -98.3141,Z 96,A -100.0148,B 24.9394,C -1.7975,E1 24.9843,E2 -174.6027} C_DIS
LIN {X -7.8211,Y -98.6053,Z 96,A -98.3318,B 24.9397,C -1.7933,E1 24.9889,E2 -176.2767} C_DIS
LIN {X -4.3081,Y -98.8211,Z 96,A -96.3835,B 24.9399,C -1.7901,E1 24.9943,E2 -178.2178} C_DIS
LIN {X -1.7598,Y -98.8993,Z 96,A -94.8171,B 24.9397,C -1.7937,E1 24.9987,E2 -179.7929} C_DIS
LIN {X 0.6782,Y -98.9101,Z 96,A -93.6564,B 24.9403,C -1.7847,E1 25.0019,E2 -180.9323} C_DIS
Enddeposition()
LIN {X 0.6782,Y -98.9101,Z 96,A -93.6564,B 24.9403,C -1.7847,E1 25.0019,E2 -180.9323} C_DIS
Startdeposition()
$VEL.CP = VEL_PRINT
LIN {X -0.4292,Y -98.0002,Z 96,A -94.9317,B 24.9408,C -1.7774,E1 24.9983,E2 -179.6398} C_DIS
LIN {X -4.0283,Y -97.9183,Z 96,A -96.9877,B 24.9407,C -1.7789,E1 24.9926,E2 -177.587} C_DIS
LIN {X -7.0845,Y -97.7458,Z 96,A -98.8591,B 24.9409,C -1.7759,E1 24.9873,E2 -175.7078} C_DIS
LIN {X -10.2664,Y -97.4618,Z 96,A -100.6629,B 24.9407,C -1.7784,E1 24.9823,E2 -173.9089} C_DIS
LIN {X -13.7562,Y -97.0307,Z 96,A -102.6935,B 24.9407,C -1.7796,E1 24.9767,E2 -171.8798} C_DIS
LIN {X -16.7877,Y -96.5541,Z 96,A -104.5699,B 24.9408,C -1.7772,E1 24.9715,E2 -169.9959} C_DIS
LIN {X -20.2874,Y -95.8799,Z 96,A -106.7148,B 24.9408,C -1.7759,E1 24.9656,E2 -167.8454} C_DIS
LIN {X -23.697,Y -95.0941,Z 96,A -108.6387,B 24.9405,C -1.7813,E1 24.9604,E2 -165.9317} C_DIS
LIN {X -26.9325,Y -94.2278,Z 96,A -110.7256,B 24.9407,C -1.778,E1 24.9548,E2 -163.8338} C_DIS
LIN {X -30.5679,Y -93.1127,Z 96,A -112.9182,B 24.9406,C -1.7807,E1 24.949,E2 -161.6438} C_DIS
LIN {X -33.9018,Y -91.951,Z 96,A -115.0147,B 24.9406,C -1.7814,E1 24.9434,E2 -159.5446} C_DIS
LIN {X -36.5291,Y -90.9397,Z 96,A -116.6897,B 24.9405,C -1.782,E1 24.9391,E2 -157.8673} C_DIS
LIN {X -39.1076,Y -89.8598,Z 96,A -119.1519,B 24.9423,C -1.7552,E1 24.9326,E2 -155.3356} C_DIS
LIN {X -43.6918,Y -87.7226,Z 96,A -121.259,B 24.9401,C -1.7879,E1 24.9275,E2 -153.3009} C_DIS
LIN {X -46.7297,Y -86.1425,Z 96,A -123.2677,B 24.9399,C -1.7903,E1 24.9226,E2 -151.2923} C_DIS
LIN {X -49.7091,Y -84.4585,Z 96,A -125.1372,B 24.9394,C -1.7977,E1 24.9181,E2 -149.4348} C_DIS
LIN {X -52.55,Y -82.7219,Z 96,A -126.9685,B 24.939,C -1.8046,E1 24.9137,E2 -147.614} C_DIS
LIN {X -55.9818,Y -80.4378,Z 96,A -130.0624,B 24.9403,C -1.7851,E1 24.9065,E2 -144.4635} C_DIS
LIN {X -58.7552,Y -78.435,Z 96,A -131.682,B 24.9392,C -1.8015,E1 24.9029,E2 -142.8771} C_DIS
LIN {X -62.1216,Y -75.7984,Z 96,A -134.1629,B 24.9388,C -1.8067,E1 24.8975,E2 -140.3994} C_DIS
LIN {X -65.1276,Y -73.2304,Z 96,A -136.3658,B 24.9383,C -1.8149,E1 24.8929,E2 -138.2073} C_DIS
LIN {X -67.3168,Y -71.2229,Z 96,A -138.3685,B 24.9386,C -1.8094,E1 24.8888,E2 -136.1834} C_DIS
LIN {X -70.3815,Y -68.1961,Z 96,A -140.7349,B 24.9379,C -1.8199,E1 24.8841,E2 -133.8318} C_DIS
LIN {X -72.9511,Y -65.4396,Z 96,A -142.8896,B 24.9375,C -1.8264,E1 24.8801,E2 -131.6832} C_DIS
LIN {X -75.8317,Y -62.0804,Z 96,A -145.5585,B 24.9373,C -1.8296,E1 24.8753,E2 -129.0097} C_DIS
LIN {X -78.0787,Y -59.2294,Z 96,A -147.7127,B 24.937,C -1.8337,E1 24.8716,E2 -126.855} C_DIS
LIN {X -79.5388,Y -57.2533,Z 96,A -149.2761,B 24.937,C -1.833,E1 24.869,E2 -125.2824} C_DIS
LIN {X -81.7772,Y -54.0064,Z 96,A -151.4554,B 24.9363,C -1.843,E1 24.8656,E2 -123.1162} C_DIS
LIN {X -83.6803,Y -51.0081,Z 96,A -153.5618,B 24.936,C -1.8475,E1 24.8625,E2 -121.0096} C_DIS
LIN {X -85.3732,Y -48.1224,Z 96,A -155.6235,B 24.9359,C -1.8492,E1 24.8597,E2 -118.9413} C_DIS
LIN {X -87.3643,Y -44.4042,Z 96,A -157.8506,B 24.9349,C -1.8639,E1 24.8568,E2 -116.7372} C_DIS
LIN {X -88.4736,Y -42.1511,Z 96,A -159.4109,B 24.9349,C -1.8649,E1 24.8549,E2 -115.171} C_DIS
LIN {X -89.7187,Y -39.4314,Z 96,A -161.1407,B 24.9344,C -1.8705,E1 24.8529,E2 -113.445} C_DIS
LIN {X -91.0012,Y -36.3766,Z 96,A -162.9877,B 24.9338,C -1.879,E1 24.851,E2 -111.6081} C_DIS
LIN {X -92.0026,Y -33.7603,Z 96,A -164.7974,B 24.9338,C -1.8782,E1 24.8492,E2 -109.7863} C_DIS
LIN {X -92.7754,Y -31.5751,Z 96,A -166.6902,B 24.9348,C -1.8648,E1 24.8475,E2 -107.8506} C_DIS
LIN {X -93.8876,Y -28.0958,Z 96,A -168.2941,B 24.9331,C -1.8884,E1 24.8462,E2 -106.2939} C_DIS
LIN {X -94.8659,Y -24.5907,Z 96,A -170.4461,B 24.9327,C -1.8941,E1 24.8446,E2 -104.143} C_DIS
LIN {X -95.633,Y -21.42,Z 96,A -172.7689,B 24.9333,C -1.8865,E1 24.8431,E2 -101.7884} C_DIS
LIN {X -96.5797,Y -16.637,Z 96,A -175.2671,B 24.9318,C -1.9068,E1 24.8419,E2 -99.3238} C_DIS
LIN {X -97.0585,Y -13.5605,Z 96,A -176.9848,B 24.9312,C -1.9159,E1 24.8412,E2 -97.6175} C_DIS
LIN {X -97.4868,Y -10.0278,Z 96,A -179.2531,B 24.9312,C -1.9164,E1 24.8405,E2 -95.3369} C_DIS
LIN {X -97.7732,Y -6.6784,Z 96,A 178.9237,B 24.9304,C -1.9272,E1 24.8401,E2 -93.5286} C_DIS
LIN {X -97.9295,Y -3.7695,Z 96,A 177.1727,B 24.9301,C -1.9311,E1 24.8399,E2 -91.7763} C_DIS
LIN {X -97.9994,Y -0.637,Z 96,A 175.3691,B 24.9296,C -1.9379,E1 24.8398,E2 -89.978} C_DIS
LIN {X -97.9614,Y 2.7949,Z 96,A 173.2474,B 24.9294,C -1.9407,E1 24.8398,E2 -87.8501} C_DIS
LIN {X -97.8029,Y 6.2393,Z 96,A 171.2837,B 24.9288,C -1.9488,E1 24.8402,E2 -85.8941} C_DIS
LIN {X -97.5747,Y 9.1315,Z 96,A 169.4897,B 24.9286,C -1.9511,E1 24.8406,E2 -84.0948} C_DIS
LIN {X -97.2219,Y 12.3354,Z 96,A 167.4642,B 24.9286,C -1.9526,E1 24.8413,E2 -82.0607} C_DIS
LIN {X -96.6812,Y 16.0302,Z 96,A 165.3344,B 24.9279,C -1.9614,E1 24.8422,E2 -79.9391} C_DIS
LIN {X -95.9575,Y 19.9095,Z 96,A 163.1131,B 24.9271,C -1.9715,E1 24.8434,E2 -77.7288} C_DIS
LIN {X -95.1749,Y 23.3656,Z 96,A 161.0325,B 24.9267,C -1.9778,E1 24.8447,E2 -75.6511} C_DIS
LIN {X -94.2493,Y 26.8568,Z 96,A 158.8659,B 24.9263,C -1.9826,E1 24.8463,E2 -73.4835} C_DIS
LIN {X -92.9545,Y 31.0441,Z 96,A 156.5805,B 24.925,C -1.9996,E1 24.8483,E2 -71.2254} C_DIS
LIN {X -91.8737,Y 34.1137,Z 96,A 154.2837,B 24.9255,C -1.9927,E1 24.8505,E2 -68.8992} C_DIS
LIN {X -90.4632,Y 37.6929,Z 96,A 152.1682,B 24.9247,C -2.0039,E1 24.8526,E2 -66.7986} C_DIS
LIN {X -89.0979,Y 40.8181,Z 96,A 150.0258,B 24.9247,C -2.0051,E1 24.8551,E2 -64.6473} C_DIS
LIN {X -87.6231,Y 43.8925,Z 96,A 148.0174,B 24.9242,C -2.0105,E1 24.8576,E2 -62.641} C_DIS
LIN {X -85.8461,Y 47.2755,Z 96,A 145.861,B 24.9235,C -2.0196,E1 24.8604,E2 -60.4947} C_DIS
LIN {X -84.3514,Y 49.8902,Z 96,A 143.9598,B 24.9235,C -2.0201,E1 24.8631,E2 -58.5849} C_DIS
LIN {X -82.6462,Y 52.6679,Z 96,A 141.773,B 24.9238,C -2.0163,E1 24.8664,E2 -56.3781} C_DIS
LIN {X -80.8307,Y 55.4158,Z 96,A 140.288,B 24.9223,C -2.036,E1 24.8687,E2 -54.9325} C_DIS
LIN {X -78.9873,Y 58.0106,Z 96,A 137.9967,B 24.923,C -2.027,E1 24.8725,E2 -52.6087} C_DIS
LIN {X -75.9153,Y 61.9773,Z 96,A 135.4009,B 24.9215,C -2.0458,E1 24.8769,E2 -50.0455} C_DIS
LIN {X -73.7679,Y 64.5175,Z 96,A 133.5843,B 24.9208,C -2.055,E1 24.8802,E2 -48.2425} C_DIS
LIN {X -71.3234,Y 67.2099,Z 96,A 131.2003,B 24.9211,C -2.0518,E1 24.8848,E2 -45.8405} C_DIS
LIN {X -68.6026,Y 69.9859,Z 96,A 129.0424,B 24.9203,C -2.061,E1 24.889,E2 -43.6954} C_DIS
LIN {X -66.1017,Y 72.3519,Z 96,A 127.0137,B 24.92,C -2.0652,E1 24.8931,E2 -41.6684} C_DIS
LIN {X -64.0563,Y 74.1707,Z 96,A 125.4542,B 24.9196,C -2.0702,E1 24.8964,E2 -40.1145} C_DIS
LIN {X -61.168,Y 76.5698,Z 96,A 123.2329,B 24.9193,C -2.0741,E1 24.9012,E2 -37.8942} C_DIS
LIN {X -58.7562,Y 78.4342,Z 96,A 121.4719,B 24.919,C -2.0786,E1 24.9051,E2 -36.1375} C_DIS
LIN {X -56.0091,Y 80.4188,Z 96,A 119.4546,B 24.9188,C -2.0814,E1 24.9097,E2 -34.1199} C_DIS
LIN {X -53.772,Y 81.9317,Z 96,A 117.6188,B 24.9192,C -2.0758,E1 24.914,E2 -32.2649} C_DIS
LIN {X -50.57,Y 83.9465,Z 96,A 115.0776,B 24.9197,C -2.0689,E1 24.9202,E2 -29.6993} C_DIS
LIN {X -47.318,Y 85.8224,Z 96,A 112.8827,B 24.9194,C -2.0727,E1 24.9255,E2 -27.5072} C_DIS
LIN {X -44.0512,Y 87.5442,Z 96,A 111.2136,B 24.9179,C -2.0926,E1 24.9296,E2 -25.881} C_DIS
LIN {X -40.6439,Y 89.1765,Z 96,A 109.0758,B 24.9174,C -2.0985,E1 24.9349,E2 -23.7518} C_DIS
LIN {X -37.8788,Y 90.3849,Z 96,A 107.3471,B 24.9171,C -2.1022,E1 24.9394,E2 -22.0279} C_DIS
LIN {X -34.7867,Y 91.6192,Z 96,A 104.4805,B 24.9194,C -2.0737,E1 24.947,E2 -19.0874} C_DIS
LIN {X -30.272,Y 93.2084,Z 96,A 102.5615,B 24.9168,C -2.1069,E1 24.9519,E2 -17.2438} C_DIS
LIN {X -25.4385,Y 94.6419,Z 96,A 99.1149,B 24.9179,C -2.0929,E1 24.9613,E2 -13.7585} C_DIS
LIN {X -22.2095,Y 95.4513,Z 96,A 97.5916,B 24.9166,C -2.1093,E1 24.9653,E2 -12.2719} C_DIS
LIN {X -18.4581,Y 96.2471,Z 96,A 95.3019,B 24.9166,C -2.1095,E1 24.9716,E2 -9.9802} C_DIS
LIN {X -15.0182,Y 96.8434,Z 96,A 93.5475,B 24.9156,C -2.1209,E1 24.9764,E2 -8.2513} C_DIS
LIN {X -12.3849,Y 97.2155,Z 96,A 91.9329,B 24.9157,C -2.1198,E1 24.9808,E2 -6.6327} C_DIS
LIN {X -9.7551,Y 97.5153,Z 96,A 90.1228,B 24.9164,C -2.1114,E1 24.9859,E2 -4.8017} C_DIS
LIN {X -6.3041,Y 97.7985,Z 96,A 88.2779,B 24.9158,C -2.1186,E1 24.991,E2 -2.9731} C_DIS
LIN {X -3.2803,Y 97.9465,Z 96,A 86.455,B 24.9159,C -2.1173,E1 24.9961,E2 -1.1468} C_DIS
LIN {X -0.6663,Y 97.9988,Z 96,A 84.7919,B 24.9163,C -2.1129,E1 25.0008,E2 0.5268} C_DIS
LIN {X 3.0437,Y 97.9537,Z 96,A 82.6541,B 24.9162,C -2.1143,E1 25.0067,E2 2.6609} C_DIS
LIN {X 6.6428,Y 97.7756,Z 96,A 80.657,B 24.9158,C -2.1182,E1 25.0123,E2 4.648} C_DIS
LIN {X 10.1664,Y 97.4723,Z 96,A 78.5838,B 24.9158,C -2.1178,E1 25.018,E2 6.7209} C_DIS
LIN {X 13.2633,Y 97.1008,Z 96,A 76.7228,B 24.916,C -2.1161,E1 25.0232,E2 8.5846} C_DIS
LIN {X 16.3594,Y 96.6261,Z 96,A 74.9517,B 24.9159,C -2.1177,E1 25.0281,E2 10.3501} C_DIS
LIN {X 19.6967,Y 96.0012,Z 96,A 72.963,B 24.9159,C -2.1167,E1 25.0335,E2 12.3388} C_DIS
LIN {X 22.1604,Y 95.4627,Z 96,A 71.3817,B 24.9163,C -2.1121,E1 25.0378,E2 13.929} C_DIS
LIN {X 26.0276,Y 94.4828,Z 96,A 69.0747,B 24.9163,C -2.1115,E1 25.0441,E2 16.2337} C_DIS
LIN {X 29.2835,Y 93.524,Z 96,A 67.1043,B 24.9165,C -2.1106,E1 25.0493,E2 18.2029} C_DIS
LIN {X 32.3316,Y 92.5142,Z 96,A 65.232,B 24.9165,C -2.1091,E1 25.0543,E2 20.0748} C_DIS
LIN {X 35.9033,Y 91.1875,Z 96,A 62.1552,B 24.9192,C -2.0761,E1 25.0625,E2 23.2229} C_DIS
LIN {X 40.4329,Y 89.2716,Z 96,A 60.0755,B 24.9171,C -2.1019,E1 25.0676,E2 25.2366} C_DIS
LIN {X 43.6253,Y 87.7556,Z 96,A 58.0174,B 24.9173,C -2.0996,E1 25.0728,E2 27.2946} C_DIS
LIN {X 46.7097,Y 86.1534,Z 96,A 56.1398,B 24.9171,C -2.1026,E1 25.0774,E2 29.1598} C_DIS
LIN {X 50.3824,Y 84.0605,Z 96,A 53.7345,B 24.9171,C -2.1015,E1 25.0832,E2 31.5605} C_DIS
LIN {X 56.354,Y 80.1791,Z 96,A 49.6377,B 24.9175,C -2.0973,E1 25.0928,E2 35.6537} C_DIS
LIN {X 59.4416,Y 77.9174,Z 96,A 47.182,B 24.9185,C -2.0852,E1 25.0983,E2 38.1293} C_DIS
LIN {X 61.7768,Y 76.0778,Z 96,A 45.5354,B 24.9185,C -2.0854,E1 25.1019,E2 39.7691} C_DIS
LIN {X 63.8895,Y 74.3136,Z 96,A 43.7723,B 24.9191,C -2.0765,E1 25.1056,E2 41.5465} C_DIS
LIN {X 66.5003,Y 71.9862,Z 96,A 41.8018,B 24.9192,C -2.0752,E1 25.1097,E2 43.5121} C_DIS
LIN {X 68.8067,Y 69.7842,Z 96,A 39.9738,B 24.9194,C -2.0727,E1 25.1133,E2 45.3384} C_DIS
LIN {X 71.4626,Y 67.0619,Z 96,A 37.7474,B 24.9198,C -2.0677,E1 25.1177,E2 47.5669} C_DIS
LIN {X 73.9666,Y 64.2899,Z 96,A 35.5375,B 24.9203,C -2.0618,E1 25.1218,E2 49.781} C_DIS
LIN {X 76.3059,Y 61.4953,Z 96,A 33.4669,B 24.9205,C -2.059,E1 25.1254,E2 51.8485} C_DIS
LIN {X 78.2772,Y 58.9652,Z 96,A 31.6747,B 24.9206,C -2.0577,E1 25.1285,E2 53.6354} C_DIS
LIN {X 80.0919,Y 56.4782,Z 96,A 29.8029,B 24.9212,C -2.0504,E1 25.1315,E2 55.5153} C_DIS
LIN {X 81.6045,Y 54.2683,Z 96,A 28.059,B 24.922,C -2.0396,E1 25.1343,E2 57.2761} C_DIS
LIN {X 83.7506,Y 50.8924,Z 96,A 26.0101,B 24.9216,C -2.0446,E1 25.1372,E2 59.3028} C_DIS
LIN {X 85.3953,Y 48.0828,Z 96,A 24.2649,B 24.9216,C -2.0456,E1 25.1397,E2 61.0367} C_DIS
LIN {X 87.252,Y 44.6238,Z 96,A 21.7394,B 24.9227,C -2.0304,E1 25.143,E2 63.5847} C_DIS
LIN {X 88.8145,Y 41.4269,Z 96,A 19.7711,B 24.9228,C -2.0289,E1 25.1453,E2 65.546} C_DIS
LIN {X 90.7121,Y 37.0882,Z 96,A 16.9736,B 24.9235,C -2.0198,E1 25.1484,E2 68.3496} C_DIS
LIN {X 91.9535,Y 33.8949,Z 96,A 14.9649,B 24.924,C -2.0137,E1 25.1504,E2 70.3615} C_DIS
LIN {X 93.5666,Y 29.1463,Z 96,A 12.0577,B 24.9246,C -2.0059,E1 25.153,E2 73.2706} C_DIS
LIN {X 94.6044,Y 25.5775,Z 96,A 9.8722,B 24.9251,C -1.9988,E1 25.1546,E2 75.4604} C_DIS
LIN {X 95.537,Y 21.8387,Z 96,A 7.6253,B 24.9256,C -1.9921,E1 25.1561,E2 77.71} C_DIS
LIN {X 96.2292,Y 18.5509,Z 96,A 5.7465,B 24.9258,C -1.9893,E1 25.1571,E2 79.5845} C_DIS
LIN {X 96.8499,Y 14.9763,Z 96,A 3.6304,B 24.9263,C -1.9829,E1 25.1581,E2 81.7034} C_DIS
LIN {X 97.3151,Y 11.576,Z 96,A 1.577,B 24.9269,C -1.9747,E1 25.1588,E2 83.7639} C_DIS
LIN {X 97.6903,Y 7.7978,Z 96,A -0.5537,B 24.9272,C -1.9711,E1 25.1594,E2 85.8905} C_DIS
LIN {X 97.8991,Y 4.4765,Z 96,A -2.4888,B 24.9276,C -1.9653,E1 25.1597,E2 87.8278} C_DIS
LIN {X 97.9913,Y 1.4312,Z 96,A -4.3481,B 24.9282,C -1.9565,E1 25.1597,E2 89.6968} C_DIS
LIN {X 97.9793,Y -2.0808,Z 96,A -6.4353,B 24.9288,C -1.9486,E1 25.1597,E2 91.7903} C_DIS
LIN {X 97.8007,Y -6.2718,Z 96,A -8.7612,B 24.929,C -1.9456,E1 25.1594,E2 94.1093} C_DIS
LIN {X 97.5423,Y -9.4826,Z 96,A -10.6106,B 24.9294,C -1.9409,E1 25.1589,E2 95.959} C_DIS
LIN {X 97.1756,Y -12.6925,Z 96,A -12.4531,B 24.9297,C -1.9366,E1 25.1583,E2 97.8005} C_DIS
LIN {X 96.719,Y -15.8036,Z 96,A -14.6195,B 24.931,C -1.9178,E1 25.1573,E2 99.9985} C_DIS
LIN {X 95.7095,Y -21.0694,Z 96,A -17.5271,B 24.9311,C -1.9167,E1 25.1557,E2 102.8918} C_DIS
LIN {X 94.7751,Y -24.9439,Z 96,A -19.6239,B 24.9311,C -1.9185,E1 25.1543,E2 104.9724} C_DIS
LIN {X 93.8868,Y -28.0984,Z 96,A -21.6796,B 24.9318,C -1.9069,E1 25.1527,E2 107.0435} C_DIS
LIN {X 92.8714,Y -31.2905,Z 96,A -23.5785,B 24.9321,C -1.9032,E1 25.1511,E2 108.9406} C_DIS
LIN {X 91.5837,Y -34.8805,Z 96,A -26.0808,B 24.9333,C -1.8856,E1 25.1486,E2 111.4704} C_DIS
LIN {X 89.8487,Y -39.1332,Z 96,A -28.9614,B 24.9345,C -1.8698,E1 25.1454,E2 114.3724} C_DIS
LIN {X 88.4256,Y -42.251,Z 96,A -30.5362,B 24.9337,C -1.8805,E1 25.1436,E2 115.9135} C_DIS
LIN {X 86.3521,Y -46.3434,Z 96,A -33.0874,B 24.9339,C -1.8776,E1 25.1403,E2 118.4579} C_DIS
LIN {X 84.8153,Y -49.0984,Z 96,A -35.0869,B 24.9347,C -1.8662,E1 25.1376,E2 120.474} C_DIS
LIN {X 82.7917,Y -52.4411,Z 96,A -37.3139,B 24.935,C -1.8619,E1 25.1343,E2 122.6999} C_DIS
LIN {X 80.9104,Y -55.2981,Z 96,A -39.2914,B 24.9353,C -1.8572,E1 25.1312,E2 124.6787} C_DIS
LIN {X 79.3584,Y -57.5037,Z 96,A -40.8633,B 24.9356,C -1.8531,E1 25.1286,E2 126.2527} C_DIS
LIN {X 77.3243,Y -60.2112,Z 96,A -42.8725,B 24.9361,C -1.8466,E1 25.1252,E2 128.2676} C_DIS
LIN {X 75.1624,Y -62.8882,Z 96,A -44.8798,B 24.9364,C -1.8415,E1 25.1217,E2 130.2777} C_DIS
LIN {X 72.8252,Y -65.5803,Z 96,A -46.7638,B 24.9363,C -1.8439,E1 25.1182,E2 132.1476} C_DIS
LIN {X 70.5339,Y -68.038,Z 96,A -48.7371,B 24.9366,C -1.8387,E1 25.1144,E2 134.1247} C_DIS
LIN {X 68.363,Y -70.2206,Z 96,A -50.611,B 24.9371,C -1.8314,E1 25.1107,E2 136.0078} C_DIS
LIN {X 65.7854,Y -72.6413,Z 96,A -52.6754,B 24.9375,C -1.8267,E1 25.1064,E2 138.075} C_DIS
LIN {X 63.4527,Y -74.6858,Z 96,A -54.5252,B 24.9378,C -1.8212,E1 25.1025,E2 139.9306} C_DIS
LIN {X 60.8305,Y -76.8365,Z 96,A -56.4873,B 24.9381,C -1.8176,E1 25.0982,E2 141.8937} C_DIS
LIN {X 58.089,Y -78.9299,Z 96,A -58.4129,B 24.9381,C -1.8168,E1 25.0939,E2 143.8142} C_DIS
LIN {X 55.6372,Y -80.6773,Z 96,A -60.1479,B 24.9383,C -1.8142,E1 25.09,E2 145.5495} C_DIS
LIN {X 53.4833,Y -82.1218,Z 96,A -61.5474,B 24.9383,C -1.8157,E1 25.0867,E2 146.9408} C_DIS
LIN {X 51.172,Y -83.5806,Z 96,A -63.3162,B 24.9389,C -1.8061,E1 25.0825,E2 148.7265} C_DIS
LIN {X 48.1225,Y -85.3731,Z 96,A -65.3891,B 24.9391,C -1.8022,E1 25.0775,E2 150.8025} C_DIS
LIN {X 45.0247,Y -87.0471,Z 96,A -67.4965,B 24.9395,C -1.7969,E1 25.0723,E2 152.9166} C_DIS
LIN {X 42.1286,Y -88.4844,Z 96,A -69.4689,B 24.9399,C -1.7907,E1 25.0673,E2 154.8983} C_DIS
LIN {X 38.9893,Y -89.9114,Z 96,A -71.7726,B 24.9408,C -1.7769,E1 25.0613,E2 157.2291} C_DIS
LIN {X 35.8105,Y -91.2239,Z 96,A -73.2586,B 24.9397,C -1.7937,E1 25.0576,E2 158.6719} C_DIS
LIN {X 32.6364,Y -92.4073,Z 96,A -75.1813,B 24.9397,C -1.7933,E1 25.0525,E2 160.5917} C_DIS
LIN {X 28.1541,Y -93.8703,Z 96,A -78.0496,B 24.9402,C -1.7858,E1 25.0449,E2 163.4725} C_DIS
LIN {X 24.9758,Y -94.7664,Z 96,A -80.0001,B 24.9404,C -1.783,E1 25.0396,E2 165.4265} C_DIS
LIN {X 21.5717,Y -95.5987,Z 96,A -82.1827,B 24.9409,C -1.7761,E1 25.0336,E2 167.6224} C_DIS
LIN {X 17.4722,Y -96.431,Z 96,A -84.4089,B 24.9405,C -1.7821,E1 25.0276,E2 169.8316} C_DIS
LIN {X 14.3989,Y -96.939,Z 96,A -86.2827,B 24.9407,C -1.7789,E1 25.0224,E2 171.7114} C_DIS
LIN {X 11.1782,Y -97.3617,Z 96,A -88.1808,B 24.9407,C -1.7777,E1 25.0171,E2 173.6107} C_DIS
LIN {X 7.9175,Y -97.6807,Z 96,A -90.1154,B 24.9409,C -1.7761,E1 25.0117,E2 175.5482} C_DIS
LIN {X 4.3267,Y -97.9055,Z 96,A -92.1393,B 24.9407,C -1.7781,E1 25.0061,E2 177.5664} C_DIS
LIN {X 1.1957,Y -97.9955,Z 96,A -94.0376,B 24.9409,C -1.7751,E1 25.0008,E2 179.4716} C_DIS
LIN {X 1.1957,Y -97.9955,Z 96,A -94.0376,B 24.9409,C -1.7751,E1 25.0008,E2 179.4716} C_DIS
Enddeposition()
LIN {X 0.6759,Y -97.0842,Z 96,A -94.2658,B 24.9397,C -1.7939,E1 25.0003,E2 179.6552} C_DIS
Startdeposition()
$VEL.CP = VEL_PRINT
LIN {X 4.3454,Y -96.9899,Z 96,A -91.2729,B 24.9376,C -1.8246,E1 25.0088,E2 176.5902} C_DIS
LIN {X 7.7275,Y -96.779,Z 96,A -89.2913,B 24.9376,C -1.8248,E1 25.0143,E2 174.6089} C_DIS
LIN {X 11.3293,Y -96.4238,Z 96,A -87.2374,B 24.9377,C -1.823,E1 25.02,E2 172.5606} C_DIS
LIN {X 14.3548,Y -96.0212,Z 96,A -85.2804,B 24.9372,C -1.83,E1 25.0255,E2 170.5888} C_DIS
LIN {X 17.7561,Y -95.4513,Z 96,A -83.1339,B 24.9368,C -1.8358,E1 25.0314,E2 168.4311} C_DIS
LIN {X 22.7373,Y -94.3875,Z 96,A -80.3041,B 24.9371,C -1.832,E1 25.0391,E2 165.6139} C_DIS
LIN {X 25.6898,Y -93.6273,Z 96,A -78.4549,B 24.9368,C -1.8358,E1 25.0441,E2 163.7588} C_DIS
LIN {X 32.0395,Y -91.6481,Z 96,A -74.7365,B 24.937,C -1.8327,E1 25.054,E2 160.0546} C_DIS
LIN {X 34.0788,Y -90.9101,Z 96,A -72.5127,B 24.9344,C -1.8702,E1 25.06,E2 157.7468} C_DIS
LIN {X 38.3939,Y -89.174,Z 96,A -70.7914,B 24.9369,C -1.8352,E1 25.0642,E2 156.1122} C_DIS
LIN {X 43.9595,Y -86.5651,Z 96,A -67.0141,B 24.9361,C -1.8466,E1 25.0738,E2 152.3178} C_DIS
LIN {X 46.7029,Y -85.1173,Z 96,A -65.0775,B 24.9356,C -1.8538,E1 25.0785,E2 150.3697} C_DIS
LIN {X 49.8745,Y -83.2991,Z 96,A -62.5552,B 24.9343,C -1.8718,E1 25.0847,E2 147.8126} C_DIS
LIN {X 54.0563,Y -80.6475,Z 96,A -60.2109,B 24.9355,C -1.8553,E1 25.0901,E2 145.5152} C_DIS
LIN {X 56.353,Y -79.0584,Z 96,A -58.4709,B 24.935,C -1.8622,E1 25.094,E2 143.7648} C_DIS
LIN {X 58.9483,Y -77.1437,Z 96,A -56.4675,B 24.9344,C -1.87,E1 25.0985,E2 141.7501} C_DIS
LIN {X 62.3348,Y -74.4339,Z 96,A -53.9759,B 24.9342,C -1.8731,E1 25.1039,E2 139.2607} C_DIS
LIN {X 64.2881,Y -72.7545,Z 96,A -52.4364,B 24.9339,C -1.8773,E1 25.1072,E2 137.7174} C_DIS
LIN {X 66.7119,Y -70.5372,Z 96,A -50.5753,B 24.9339,C -1.8789,E1 25.111,E2 135.8601} C_DIS
LIN {X 69.1594,Y -68.1387,Z 96,A -48.4076,B 24.9331,C -1.8895,E1 25.1153,E2 133.6766} C_DIS
LIN {X 72.0235,Y -65.1054,Z 96,A -46.2963,B 24.9336,C -1.882,E1 25.1192,E2 131.5922} C_DIS
LIN {X 73.6227,Y -63.2912,Z 96,A -44.6703,B 24.9328,C -1.8934,E1 25.1222,E2 129.9466} C_DIS
LIN {X 75.6246,Y -60.8845,Z 96,A -42.8907,B 24.9326,C -1.8956,E1 25.1254,E2 128.17} C_DIS
LIN {X 77.9267,Y -57.9096,Z 96,A -40.1105,B 24.9306,C -1.9236,E1 25.1301,E2 125.337} C_DIS
LIN {X 80.0362,Y -54.9581,Z 96,A -38.7059,B 24.9323,C -1.9006,E1 25.1323,E2 123.9935} C_DIS
LIN {X 82.0132,Y -51.962,Z 96,A -36.3453,B 24.9312,C -1.9161,E1 25.1359,E2 121.6083} C_DIS
LIN {X 83.749,Y -49.1133,Z 96,A -34.3699,B 24.9307,C -1.922,E1 25.1387,E2 119.629} C_DIS
LIN {X 86.4363,Y -44.2116,Z 96,A -31.0443,B 24.93,C -1.9328,E1 25.1431,E2 116.2955} C_DIS
LIN {X 87.668,Y -41.7175,Z 96,A -28.8228,B 24.9279,C -1.9607,E1 25.1459,E2 114.0202} C_DIS
LIN {X 89.4174,Y -37.8213,Z 96,A -27.4094,B 24.9306,C -1.9246,E1 25.1473,E2 112.6996} C_DIS
LIN {X 90.335,Y -35.5737,Z 96,A -25.2639,B 24.9282,C -1.9571,E1 25.1496,E2 110.4894} C_DIS
LIN {X 91.993,Y -31.0352,Z 96,A -22.7855,B 24.9286,C -1.9512,E1 25.1519,E2 108.0389} C_DIS
LIN {X 93.8708,Y -24.7887,Z 96,A -19.0852,B 24.9282,C -1.9573,E1 25.1548,E2 104.3451} C_DIS
LIN {X 94.5124,Y -22.2134,Z 96,A -17.1696,B 24.9268,C -1.9761,E1 25.156,E2 102.3963} C_DIS
LIN {X 95.3698,Y -18.1805,Z 96,A -15.028,B 24.9271,C -1.9724,E1 25.1572,E2 100.2759} C_DIS
LIN {X 95.7996,Y -15.7606,Z 96,A -13.4919,B 24.9265,C -1.9804,E1 25.1579,E2 98.73} C_DIS
LIN {X 96.3026,Y -12.318,Z 96,A -11.5,B 24.9262,C -1.9846,E1 25.1587,E2 96.7399} C_DIS
LIN {X 96.6812,Y -8.8679,Z 96,A -9.5231,B 24.9259,C -1.9884,E1 25.1592,E2 94.7658} C_DIS
LIN {X 96.9444,Y -5.2629,Z 96,A -7.3029,B 24.9251,C -1.9987,E1 25.1596,E2 92.5344} C_DIS
LIN {X 97.0642,Y -2.1336,Z 96,A -5.4932,B 24.9248,C -2.0031,E1 25.1598,E2 90.7251} C_DIS
LIN {X 97.0793,Y 1.3134,Z 96,A -3.4856,B 24.9244,C -2.0086,E1 25.1598,E2 88.7165} C_DIS
LIN {X 96.9938,Y 4.2548,Z 96,A -1.7214,B 24.9238,C -2.0153,E1 25.1596,E2 86.947} C_DIS
LIN {X 96.7716,Y 7.821,Z 96,A 0.2959,B 24.9236,C -2.0184,E1 25.1592,E2 84.9343} C_DIS
LIN {X 96.4287,Y 11.2869,Z 96,A 2.3314,B 24.9232,C -2.0241,E1 25.1585,E2 82.8974} C_DIS
LIN {X 95.9557,Y 14.7785,Z 96,A 4.4093,B 24.9227,C -2.0306,E1 25.1577,E2 80.8163} C_DIS
LIN {X 95.3486,Y 18.2908,Z 96,A 6.4812,B 24.9223,C -2.036,E1 25.1567,E2 78.744} C_DIS
LIN {X 94.4812,Y 22.3485,Z 96,A 8.826,B 24.922,C -2.0395,E1 25.1553,E2 76.4046} C_DIS
LIN {X 93.783,Y 25.1135,Z 96,A 10.6661,B 24.9211,C -2.0508,E1 25.154,E2 74.5483} C_DIS
LIN {X 92.4717,Y 29.5802,Z 96,A 13.6656,B 24.9197,C -2.069,E1 25.1515,E2 71.5231} C_DIS
LIN {X 90.5633,Y 34.9922,Z 96,A 16.5522,B 24.9205,C -2.0593,E1 25.1488,E2 68.6753} C_DIS
LIN {X 88.639,Y 39.6121,Z 96,A 19.6781,B 24.9193,C -2.0745,E1 25.1453,E2 65.5307} C_DIS
LIN {X 87.154,Y 42.7811,Z 96,A 21.8576,B 24.9185,C -2.0848,E1 25.1427,E2 63.3387} C_DIS
LIN {X 84.7099,Y 47.4357,Z 96,A 25.2542,B 24.9169,C -2.1047,E1 25.1381,E2 59.9129} C_DIS
LIN {X 83.018,Y 50.338,Z 96,A 27.489,B 24.9157,C -2.1198,E1 25.1348,E2 57.6538} C_DIS
LIN {X 80.6607,Y 54.0369,Z 96,A 29.1504,B 24.918,C -2.0904,E1 25.1324,E2 56.0701} C_DIS
LIN {X 78.3873,Y 57.2829,Z 96,A 31.7873,B 24.9167,C -2.1078,E1 25.1281,E2 53.405} C_DIS
LIN {X 76.1707,Y 60.199,Z 96,A 33.7482,B 24.9169,C -2.1053,E1 25.1247,E2 51.4592} C_DIS
LIN {X 73.9426,Y 62.9158,Z 96,A 35.8682,B 24.9164,C -2.1119,E1 25.1209,E2 49.3333} C_DIS
LIN {X 70.9065,Y 66.3192,Z 96,A 38.5726,B 24.9158,C -2.1184,E1 25.1159,E2 46.6255} C_DIS
LIN {X 68.6353,Y 68.6688,Z 96,A 40.5942,B 24.9152,C -2.1261,E1 25.1119,E2 44.5944} C_DIS
LIN {X 65.828,Y 71.3627,Z 96,A 43.277,B 24.9137,C -2.1456,E1 25.1063,E2 41.8765} C_DIS
LIN {X 63.1693,Y 73.7266,Z 96,A 44.8624,B 24.9149,C -2.1301,E1 25.1031,E2 40.3339} C_DIS
LIN {X 60.3638,Y 76.0404,Z 96,A 47.0036,B 24.9146,C -2.1339,E1 25.0984,E2 38.1917} C_DIS
LIN {X 57.3143,Y 78.3643,Z 96,A 49.1683,B 24.9146,C -2.1342,E1 25.0936,E2 36.0341} C_DIS
LIN {X 51.6025,Y 82.2382,Z 96,A 53.2788,B 24.9139,C -2.1421,E1 25.084,E2 31.9186} C_DIS
LIN {X 48.6514,Y 84.0181,Z 96,A 55.4753,B 24.9132,C -2.1512,E1 25.0787,E2 29.7074} C_DIS
LIN {X 45.9494,Y 85.526,Z 96,A 57.1154,B 24.9136,C -2.1467,E1 25.0747,E2 28.0826} C_DIS
LIN {X 43.0925,Y 86.9996,Z 96,A 58.9914,B 24.9134,C -2.1484,E1 25.0701,E2 26.2078} C_DIS
LIN {X 40.2828,Y 88.3367,Z 96,A 61.4912,B 24.9113,C -2.1752,E1 25.0636,E2 23.6508} C_DIS
LIN {X 36.7223,Y 89.8743,Z 96,A 63.1284,B 24.913,C -2.1534,E1 25.0595,E2 22.069} C_DIS
LIN {X 33.8639,Y 90.9914,Z 96,A 65.4913,B 24.9112,C -2.1755,E1 25.0532,E2 19.6589} C_DIS
LIN {X 30.4752,Y 92.1818,Z 96,A 66.9574,B 24.913,C -2.1532,E1 25.0495,E2 18.2485} C_DIS
LIN {X 27.982,Y 92.968,Z 96,A 68.6541,B 24.9125,C -2.16,E1 25.0449,E2 16.5387} C_DIS
LIN {X 24.5793,Y 93.9252,Z 96,A 71.1296,B 24.9112,C -2.1756,E1 25.0381,E2 14.0302} C_DIS
LIN {X 21.4652,Y 94.6853,Z 96,A 72.5531,B 24.9125,C -2.1595,E1 25.0344,E2 12.6467} C_DIS
LIN {X 17.9424,Y 95.4156,Z 96,A 74.5985,B 24.9127,C -2.1576,E1 25.0288,E2 10.6082} C_DIS
LIN {X 14.9426,Y 95.9303,Z 96,A 76.5083,B 24.9123,C -2.1623,E1 25.0235,E2 8.6893} C_DIS
LIN {X 11.4787,Y 96.4063,Z 96,A 78.56,B 24.9123,C -2.1623,E1 25.0178,E2 6.6391} C_DIS
LIN {X 8.1838,Y 96.7426,Z 96,A 80.572,B 24.9121,C -2.1646,E1 25.0122,E2 4.623} C_DIS
LIN {X 4.65,Y 96.9768,Z 96,A 82.6584,B 24.9121,C -2.1644,E1 25.0064,E2 2.5378} C_DIS
LIN {X 1.2471,Y 97.0805,Z 96,A 85.138,B 24.9108,C -2.1809,E1 24.9994,E2 0.0193} C_DIS
LIN {X -2.2583,Y 97.0619,Z 96,A 86.7929,B 24.912,C -2.1657,E1 24.9948,E2 -1.5995} C_DIS
LIN {X -5.7476,Y 96.9176,Z 96,A 88.7419,B 24.9124,C -2.161,E1 24.9894,E2 -3.5378} C_DIS
LIN {X -9.2699,Y 96.6441,Z 96,A 91.0894,B 24.9117,C -2.1692,E1 24.9828,E2 -5.9061} C_DIS
LIN {X -13.0901,Y 96.2022,Z 96,A 93.3204,B 24.912,C -2.1665,E1 24.9767,E2 -8.1322} C_DIS
LIN {X -16.9153,Y 95.6025,Z 96,A 95.4031,B 24.9127,C -2.1578,E1 24.971,E2 -10.1961} C_DIS
LIN {X -20.2619,Y 94.9502,Z 96,A 97.8669,B 24.9115,C -2.1718,E1 24.9642,E2 -12.6963} C_DIS
LIN {X -23.4264,Y 94.219,Z 96,A 99.4164,B 24.9127,C -2.1572,E1 24.96,E2 -14.2133} C_DIS
LIN {X -27.9111,Y 92.989,Z 96,A 102.2044,B 24.9128,C -2.1558,E1 24.9526,E2 -17.0023} C_DIS
LIN {X -31.4007,Y 91.8698,Z 96,A 104.7217,B 24.912,C -2.1654,E1 24.9458,E2 -19.5473} C_DIS
LIN {X -34.4845,Y 90.7564,Z 96,A 106.1768,B 24.9136,C -2.1464,E1 24.9421,E2 -20.9601} C_DIS
LIN {X -37.5707,Y 89.523,Z 96,A 108.1508,B 24.9138,C -2.144,E1 24.937,E2 -22.933} C_DIS
LIN {X -40.4966,Y 88.2394,Z 96,A 110.4848,B 24.9128,C -2.1565,E1 24.931,E2 -25.3024} C_DIS
LIN {X -44.053,Y 86.5173,Z 96,A 113.2644,B 24.9118,C -2.1681,E1 24.924,E2 -28.1171} C_DIS
LIN {X -48.2716,Y 84.2363,Z 96,A 115.4118,B 24.9141,C -2.1398,E1 24.9189,E2 -30.2034} C_DIS
LIN {X -51.3489,Y 82.3966,Z 96,A 118.141,B 24.9128,C -2.1567,E1 24.9124,E2 -32.9814} C_DIS
LIN {X -55.1104,Y 79.9304,Z 96,A 120.3022,B 24.9145,C -2.1347,E1 24.9075,E2 -35.0975} C_DIS
LIN {X -58.7439,Y 77.3003,Z 96,A 122.7563,B 24.9155,C -2.1227,E1 24.902,E2 -37.5317} C_DIS
LIN {X -63.1351,Y 73.7557,Z 96,A 126.2196,B 24.9157,C -2.1199,E1 24.8945,E2 -41.0014} C_DIS
LIN {X -66.3057,Y 70.9192,Z 96,A 128.5987,B 24.9165,C -2.1097,E1 24.8897,E2 -43.3658} C_DIS
LIN {X -68.805,Y 68.4975,Z 96,A 131.2451,B 24.9153,C -2.1245,E1 24.8844,E2 -46.0587} C_DIS
LIN {X -71.4724,Y 65.7084,Z 96,A 132.9295,B 24.9174,C -2.0991,E1 24.8813,E2 -47.6899} C_DIS
LIN {X -74.9396,Y 61.7262,Z 96,A 136.1226,B 24.9178,C -2.0936,E1 24.8755,E2 -50.8845} C_DIS
LIN {X -77.2085,Y 58.8642,Z 96,A 138.7617,B 24.917,C -2.1039,E1 24.8709,E2 -53.5607} C_DIS
LIN {X -79.3574,Y 55.934,Z 96,A 140.9425,B 24.9174,C -2.0992,E1 24.8674,E2 -55.7411} C_DIS
LIN {X -81.4238,Y 52.8802,Z 96,A 142.7355,B 24.9188,C -2.0804,E1 24.8647,E2 -57.4984} C_DIS
LIN {X -84.7647,Y 47.3375,Z 96,A 146.3921,B 24.9201,C -2.0641,E1 24.8596,E2 -61.1349} C_DIS
LIN {X -87.1914,Y 42.7056,Z 96,A 149.4809,B 24.9208,C -2.0551,E1 24.8556,E2 -64.2188} C_DIS
LIN {X -88.551,Y 39.8073,Z 96,A 151.4301,B 24.9211,C -2.0514,E1 24.8533,E2 -66.1697} C_DIS
LIN {X -89.9649,Y 36.4997,Z 96,A 153.4718,B 24.9218,C -2.0423,E1 24.8512,E2 -68.201} C_DIS
LIN {X -91.7624,Y 31.7137,Z 96,A 156.56,B 24.9223,C -2.0353,E1 24.8482,E2 -71.2899} C_DIS
LIN {X -93.3558,Y 26.6576,Z 96,A 159.4043,B 24.9238,C -2.0163,E1 24.8459,E2 -74.1052} C_DIS
LIN {X -94.3244,Y 22.9957,Z 96,A 161.9725,B 24.9235,C -2.02,E1 24.8441,E2 -76.6972} C_DIS
LIN {X -95.0781,Y 19.6487,Z 96,A 164.56,B 24.9226,C -2.0319,E1 24.8425,E2 -79.3285} C_DIS
LIN {X -95.7338,Y 16.154,Z 96,A 166.0528,B 24.9246,C -2.0054,E1 24.8419,E2 -80.7669} C_DIS
LIN {X -96.3782,Y 11.7186,Z 96,A 168.6103,B 24.9254,C -1.9941,E1 24.8409,E2 -83.3126} C_DIS
LIN {X -96.6915,Y 8.7561,Z 96,A 170.5502,B 24.9254,C -1.9943,E1 24.8403,E2 -85.2647} C_DIS
LIN {X -96.9838,Y 4.4878,Z 96,A 173.1611,B 24.9258,C -1.989,E1 24.8399,E2 -87.8786} C_DIS
LIN {X -97.0677,Y 1.9439,Z 96,A 174.6043,B 24.9263,C -1.9823,E1 24.8398,E2 -89.3145} C_DIS
LIN {X -97.0745,Y -1.5741,Z 96,A 176.7314,B 24.9267,C -1.9772,E1 24.8398,E2 -91.4425} C_DIS
LIN {X -96.9685,Y -4.8265,Z 96,A 178.7508,B 24.9269,C -1.9743,E1 24.8401,E2 -93.4669} C_DIS
LIN {X -96.7242,Y -8.4018,Z 96,A -179.3391,B 24.9279,C -1.9609,E1 24.8405,E2 -95.3565} C_DIS
LIN {X -96.445,Y -11.1477,Z 96,A -177.5888,B 24.9279,C -1.9597,E1 24.841,E2 -97.1146} C_DIS
LIN {X -96.0315,Y -14.2884,Z 96,A -175.3457,B 24.9275,C -1.966,E1 24.8419,E2 -99.3861} C_DIS
LIN {X -95.3657,Y -18.2017,Z 96,A -172.2931,B 24.9263,C -1.9823,E1 24.8436,E2 -102.4955} C_DIS
LIN {X -94.1945,Y -23.5278,Z 96,A -170.2152,B 24.9298,C -1.9346,E1 24.8448,E2 -104.4719} C_DIS
LIN {X -93.0536,Y -27.6934,Z 96,A -167.025,B 24.9289,C -1.9481,E1 24.8473,E2 -107.7126} C_DIS
LIN {X -92.0144,Y -30.9716,Z 96,A -165.6085,B 24.9308,C -1.9218,E1 24.8485,E2 -109.0745} C_DIS
LIN {X -91.0115,Y -33.8104,Z 96,A -163.2113,B 24.9297,C -1.937,E1 24.8509,E2 -111.5216} C_DIS
LIN {X -89.8072,Y -36.8872,Z 96,A -161.7533,B 24.9312,C -1.9151,E1 24.8524,E2 -112.9354} C_DIS
LIN {X -88.5286,Y -39.857,Z 96,A -159.8707,B 24.9317,C -1.9088,E1 24.8545,E2 -114.8134} C_DIS
LIN {X -87.1766,Y -42.7355,Z 96,A -157.8667,B 24.9317,C -1.9077,E1 24.8569,E2 -116.8257} C_DIS
LIN {X -84.6475,Y -47.5473,Z 96,A -154.6535,B 24.9324,C -1.8992,E1 24.8612,E2 -120.0355} C_DIS
LIN {X -82.7161,Y -50.8347,Z 96,A -152.3766,B 24.9327,C -1.8941,E1 24.8644,E2 -122.3121} C_DIS
LIN {X -80.9404,Y -53.6151,Z 96,A -150.4898,B 24.9332,C -1.8871,E1 24.8673,E2 -124.1916} C_DIS
LIN {X -77.8461,Y -58.0174,Z 96,A -147.0687,B 24.9332,C -1.8874,E1 24.8729,E2 -127.6302} C_DIS
LIN {X -75.919,Y -60.5174,Z 96,A -145.3679,B 24.9339,C -1.8775,E1 24.8758,E2 -129.3154} C_DIS
LIN {X -71.3656,Y -65.8249,Z 96,A -141.4221,B 24.935,C -1.862,E1 24.883,E2 -133.242} C_DIS
LIN {X -69.4734,Y -67.8209,Z 96,A -138.8842,B 24.9331,C -1.8896,E1 24.8881,E2 -135.8567} C_DIS
LIN {X -66.4264,Y -70.8057,Z 96,A -137.2148,B 24.9355,C -1.8555,E1 24.8913,E2 -137.4517} C_DIS
LIN {X -64.2725,Y -72.7684,Z 96,A -134.9035,B 24.9343,C -1.8723,E1 24.8963,E2 -139.8122} C_DIS
LIN {X -61.7772,Y -74.8972,Z 96,A -133.7402,B 24.9364,C -1.8422,E1 24.8986,E2 -140.9083} C_DIS
LIN {X -59.5202,Y -76.703,Z 96,A -131.6753,B 24.9357,C -1.8514,E1 24.9032,E2 -143.0027} C_DIS
LIN {X -53.5495,Y -80.9837,Z 96,A -127.4459,B 24.9365,C -1.8404,E1 24.9128,E2 -147.2205} C_DIS
LIN {X -51.1741,Y -82.5058,Z 96,A -125.5099,B 24.936,C -1.8473,E1 24.9175,E2 -149.1789} C_DIS
LIN {X -48.0656,Y -84.3547,Z 96,A -123.4633,B 24.9365,C -1.8412,E1 24.9224,E2 -151.2173} C_DIS
LIN {X -45.1057,Y -85.9732,Z 96,A -121.509,B 24.9367,C -1.8373,E1 24.9272,E2 -153.1677} C_DIS
LIN {X -39.9694,Y -88.478,Z 96,A -118.1074,B 24.9369,C -1.8344,E1 24.9358,E2 -156.571} C_DIS
LIN {X -36.5783,Y -89.9329,Z 96,A -115.4939,B 24.936,C -1.8476,E1 24.9426,E2 -159.2217} C_DIS
LIN {X -33.3691,Y -91.1724,Z 96,A -114.0356,B 24.9375,C -1.8255,E1 24.9463,E2 -160.6305} C_DIS
LIN {X -30.5544,Y -92.1551,Z 96,A -112.1254,B 24.9373,C -1.8293,E1 24.9514,E2 -162.5535} C_DIS
LIN {X -27.486,Y -93.1151,Z 96,A -109.8878,B 24.9365,C -1.8402,E1 24.9574,E2 -164.8206} C_DIS
LIN {X -23.3591,Y -94.2358,Z 96,A -107.6986,B 24.9375,C -1.8267,E1 24.9633,E2 -166.981} C_DIS
LIN {X -20.2035,Y -94.963,Z 96,A -105.7658,B 24.9375,C -1.8266,E1 24.9686,E2 -168.9159} C_DIS
LIN {X -16.9468,Y -95.5969,Z 96,A -103.8326,B 24.9375,C -1.825,E1 24.9739,E2 -170.8474} C_DIS
LIN {X -13.4031,Y -96.1578,Z 96,A -101.6852,B 24.9375,C -1.8256,E1 24.9798,E2 -172.998} C_DIS
LIN {X -9.63,Y -96.6095,Z 96,A -99.4306,B 24.9375,C -1.8257,E1 24.9861,E2 -175.2543} C_DIS
LIN {X -5.9824,Y -96.9042,Z 96,A -97.2944,B 24.9375,C -1.8249,E1 24.992,E2 -177.3893} C_DIS
LIN {X -2.792,Y -97.0471,Z 96,A -95.398,B 24.9375,C -1.8256,E1 24.9973,E2 -179.2876} C_DIS
LIN {X 0.6759,Y -97.0842,Z 96,A -94.2634,B 24.9398,C -1.7929,E1 25.0003,E2 -180.3448} C_DIS
Enddeposition()
LIN {X 0.6759,Y -97.0842,Z 96,A -94.2634,B 24.9398,C -1.7929,E1 25.0003,E2 -180.3448} C_DIS
Startdeposition()
$VEL.CP = VEL_PRINT
LIN {X 0.0215,Y -96.1748,Z 96,A -94.8007,B 24.939,C -1.8036,E1 24.9988,E2 -179.833} C_DIS
LIN {X -3.2605,Y -96.1183,Z 96,A -96.7949,B 24.9391,C -1.802,E1 24.9933,E2 -177.8346} C_DIS
LIN {X -6.7788,Y -95.9344,Z 96,A -98.8508,B 24.9391,C -1.8034,E1 24.9875,E2 -175.7814} C_DIS
LIN {X -10.1907,Y -95.6318,Z 96,A -100.9152,B 24.9391,C -1.8028,E1 24.9818,E2 -173.7144} C_DIS
LIN {X -13.8025,Y -95.1779,Z 96,A -103.0294,B 24.9389,C -1.8051,E1 24.976,E2 -171.6041} C_DIS
LIN {X -17.27,Y -94.6101,Z 96,A -105.1925,B 24.939,C -1.8033,E1 24.97,E2 -169.4346} C_DIS
LIN {X -20.6589,Y -93.9282,Z 96,A -107.3852,B 24.9393,C -1.7996,E1 24.964,E2 -167.2306} C_DIS
LIN {X -23.8362,Y -93.1725,Z 96,A -109.8788,B 24.9405,C -1.7819,E1 24.9571,E2 -164.6912} C_DIS
LIN {X -28.1,Y -91.9773,Z 96,A -111.7883,B 24.9387,C -1.8087,E1 24.9522,E2 -162.8422} C_DIS
LIN {X -32.597,Y -90.4812,Z 96,A -114.9281,B 24.9393,C -1.8002,E1 24.9438,E2 -159.6762} C_DIS
LIN {X -36.8626,Y -88.8296,Z 96,A -117.189,B 24.938,C -1.8187,E1 24.938,E2 -157.4543} C_DIS
LIN {X -40.8495,Y -87.0668,Z 96,A -120.2651,B 24.9389,C -1.8054,E1 24.9301,E2 -154.3389} C_DIS
LIN {X -44.992,Y -85.0002,Z 96,A -122.754,B 24.9381,C -1.8179,E1 24.924,E2 -151.8731} C_DIS
LIN {X -47.7006,Y -83.5104,Z 96,A -124.7254,B 24.9381,C -1.8161,E1 24.9192,E2 -149.8916} C_DIS
LIN {X -50.9925,Y -81.5416,Z 96,A -126.7443,B 24.9373,C -1.8284,E1 24.9144,E2 -147.8959} C_DIS
LIN {X -53.8826,Y -79.6614,Z 96,A -129.6756,B 24.9391,C -1.8025,E1 24.9075,E2 -144.8931} C_DIS
LIN {X -57.543,Y -77.0594,Z 96,A -131.607,B 24.9371,C -1.8318,E1 24.9033,E2 -143.0245} C_DIS
LIN {X -60.7335,Y -74.5705,Z 96,A -134.1016,B 24.937,C -1.8334,E1 24.8978,E2 -140.5244} C_DIS
LIN {X -63.8577,Y -71.9139,Z 96,A -136.4831,B 24.9365,C -1.8401,E1 24.8928,E2 -138.1497} C_DIS
LIN {X -67.8155,Y -68.1941,Z 96,A -139.8702,B 24.9365,C -1.8418,E1 24.8859,E2 -134.7526} C_DIS
LIN {X -69.7947,Y -66.1673,Z 96,A -141.5051,B 24.936,C -1.8472,E1 24.8828,E2 -133.1234} C_DIS
LIN {X -73.9446,Y -61.4936,Z 96,A -145.1272,B 24.9352,C -1.859,E1 24.8762,E2 -129.5131} C_DIS
LIN {X -76.078,Y -58.8339,Z 96,A -147.0799,B 24.9347,C -1.8664,E1 24.8728,E2 -127.5689} C_DIS
LIN {X -77.7055,Y -56.6671,Z 96,A -149.2124,B 24.9356,C -1.8536,E1 24.8692,E2 -125.3954} C_DIS
LIN {X -80.4265,Y -52.7343,Z 96,A -151.6636,B 24.9342,C -1.8737,E1 24.8654,E2 -122.9799} C_DIS
LIN {X -81.8576,Y -50.4866,Z 96,A -153.3458,B 24.9342,C -1.8747,E1 24.8629,E2 -121.2916} C_DIS
LIN {X -83.6291,Y -47.4939,Z 96,A -155.2028,B 24.9332,C -1.8872,E1 24.8603,E2 -119.4548} C_DIS
LIN {X -84.7929,Y -45.3836,Z 96,A -157.4191,B 24.9347,C -1.8661,E1 24.8574,E2 -117.1763} C_DIS
LIN {X -86.5401,Y -41.9546,Z 96,A -159.1045,B 24.9329,C -1.8918,E1 24.8553,E2 -115.5433} C_DIS
LIN {X -88.0106,Y -38.7756,Z 96,A -161.1096,B 24.9323,C -1.9004,E1 24.853,E2 -113.5475} C_DIS
LIN {X -90.0606,Y -33.7413,Z 96,A -164.5386,B 24.9321,C -1.9037,E1 24.8495,E2 -110.1072} C_DIS
LIN {X -91.1942,Y -30.5438,Z 96,A -166.7918,B 24.9321,C -1.9023,E1 24.8474,E2 -107.838} C_DIS
LIN {X -92.9968,Y -24.5192,Z 96,A -170.2855,B 24.9308,C -1.9216,E1 24.8448,E2 -104.3702} C_DIS
LIN {X -93.9078,Y -20.7522,Z 96,A -172.9809,B 24.9311,C -1.9165,E1 24.8431,E2 -101.6467} C_DIS
LIN {X -94.5847,Y -17.4113,Z 96,A -175.2169,B 24.9311,C -1.9164,E1 24.8419,E2 -99.3972} C_DIS
LIN {X -95.1833,Y -13.7649,Z 96,A -176.8541,B 24.9294,C -1.9411,E1 24.8413,E2 -97.8091} C_DIS
LIN {X -95.6067,Y -10.4312,Z 96,A -178.7487,B 24.9287,C -1.9508,E1 24.8406,E2 -95.9264} C_DIS
LIN {X -95.9484,Y -6.5714,Z 96,A 178.4439,B 24.9293,C -1.9424,E1 24.84,E2 -93.0822} C_DIS
LIN {X -96.1564,Y -1.7953,Z 96,A 175.9609,B 24.9278,C -1.963,E1 24.8398,E2 -90.6334} C_DIS
LIN {X -96.1584,Y 1.6829,Z 96,A 173.5769,B 24.928,C -1.9599,E1 24.8398,E2 -88.2275} C_DIS
LIN {X -95.8448,Y 7.9453,Z 96,A 170.0039,B 24.9267,C -1.977,E1 24.8405,E2 -84.6738} C_DIS
LIN {X -95.5919,Y 10.5708,Z 96,A 167.6858,B 24.9281,C -1.9587,E1 24.8412,E2 -82.2981} C_DIS
LIN {X -94.9835,Y 15.0852,Z 96,A 165.9702,B 24.9251,C -1.9986,E1 24.8419,E2 -80.6677} C_DIS
LIN {X -93.8956,Y 20.8084,Z 96,A 162.2071,B 24.925,C -2.0004,E1 24.8439,E2 -76.8866} C_DIS
LIN {X -93.2166,Y 23.6648,Z 96,A 159.7285,B 24.9263,C -1.9831,E1 24.8457,E2 -74.3523} C_DIS
LIN {X -92.0113,Y 27.9891,Z 96,A 157.7234,B 24.9241,C -2.0124,E1 24.8472,E2 -72.4055} C_DIS
LIN {X -90.8754,Y 31.4813,Z 96,A 155.4242,B 24.9238,C -2.0157,E1 24.8493,E2 -70.101} C_DIS
LIN {X -89.3097,Y 35.6842,Z 96,A 152.8461,B 24.923,C -2.0269,E1 24.8519,E2 -67.535} C_DIS
LIN {X -87.9775,Y 38.8515,Z 96,A 150.7964,B 24.9225,C -2.033,E1 24.8541,E2 -65.4887} C_DIS
LIN {X -86.7553,Y 41.5067,Z 96,A 148.6028,B 24.9232,C -2.024,E1 24.8568,E2 -63.2616} C_DIS
LIN {X -85.1958,Y 44.6205,Z 96,A 147.0413,B 24.9215,C -2.0463,E1 24.8587,E2 -61.745} C_DIS
LIN {X -83.6065,Y 47.5327,Z 96,A 144.6068,B 24.9222,C -2.0375,E1 24.8621,E2 -59.2767} C_DIS
LIN {X -81.714,Y 50.7165,Z 96,A 142.481,B 24.9215,C -2.0463,E1 24.8652,E2 -57.1611} C_DIS
LIN {X -78.6765,Y 55.3131,Z 96,A 138.6925,B 24.922,C -2.0394,E1 24.8713,E2 -53.3373} C_DIS
Enddeposition()
END
